	    //PathData - command - cmdParameters - bufferMode
	    IF #tempPathDataCmd_checking.cmdParameters.bufferMode <> "BM_BUFFERED"
	      AND #tempPathDataCmd_checking.cmdParameters.bufferMode <> "BM_BLENDING_LOW"
	      AND #tempPathDataCmd_checking.cmdParameters.bufferMode <> "BM_BLENDING_HIGH"
	    THEN
	      #LKinCtrl_CheckPathDataCmd := #ERR_PATHDATA_BUFFERMODE;
	      RETURN;
	    END_IF;
	    
	    //PathData - command - cmdParameters - dynamicAdaption
	    IF #tempPathDataCmd_checking.cmdParameters.dynamicAdaption > "DA_WITH_CONSTANT_LIMITS"
	    THEN
	      #LKinCtrl_CheckPathDataCmd := #ERR_PATHDATA_DYNAMICADAPTION;
	      RETURN;
	    END_IF;
	    
	    //PathData - command - setFlags
	    FOR #tempFlagCtr := 1 TO "LKINCTRL_NO_OF_CMD_SETFLAGS" DO
	      // check flag to be in range of flags InOut array at LKinCtrl_MC_MovePath
	      IF #tempPathDataCmd_checking.setFlags[#tempFlagCtr].flag <> -1
	        AND (#tempPathDataCmd_checking.setFlags[#tempFlagCtr].flag < #firstFlag OR #tempPathDataCmd_checking.setFlags[#tempFlagCtr].flag > #lastFlag)
	      THEN
	        #LKinCtrl_CheckPathDataCmd := #ERR_PATHDATA_SETFLAGS_FLAG;
	        RETURN;
	      END_IF;
	      
	      // check flagMode to be valid
	      IF "LKinCtrl_CheckFlagMode"(#tempPathDataCmd_checking.setFlags[#tempFlagCtr].flagMode) = FALSE THEN
	        #LKinCtrl_CheckPathDataCmd := #ERR_PATHDATA_SETFLAGS_FLAGMODE;
	        RETURN;
	      END_IF;
	    END_FOR;
	    
	    //PathData - command - valueFlags
	    FOR #tempFlagCtr := 1 TO "LKINCTRL_NO_OF_CMD_VALUEFLAGS" DO
	      // check flag to be in range of flags InOut array at LKinCtrl_MC_MovePath
	      IF #tempPathDataCmd_checking.valueFlags[#tempFlagCtr].flag <> -1
	        AND (#tempPathDataCmd_checking.valueFlags[#tempFlagCtr].flag < #firstFlag OR #tempPathDataCmd_checking.valueFlags[#tempFlagCtr].flag > #lastFlag)
	      THEN
	        #LKinCtrl_CheckPathDataCmd := #ERR_PATHDATA_VALUEFLAGS_FLAG;
	        RETURN;
	      END_IF;
	      
	      // check flagMode to be valid
	      IF "LKinCtrl_CheckFlagMode"(#tempPathDataCmd_checking.valueFlags[#tempFlagCtr].flagMode) = FALSE THEN
	        #LKinCtrl_CheckPathDataCmd := #ERR_PATHDATA_VALUEFLAGS_FLAGMODE;
	        RETURN;
	      END_IF;
	    END_FOR;
	  END_REGION
	END_REGION CHECK_COMMAND
	
	
END_FUNCTION

FUNCTION "LKinCtrl_CheckFlagMode" : Bool
TITLE = LKinCtrl_CheckFlagMode
{ S7_Optimized_Access := 'TRUE' }
AUTHOR : 'handling.team.automation@siemens.com'
FAMILY : LKinCtrl
VERSION : 5.0
//Check given flag mode to be valid
   VAR_INPUT 
      flagMode : DInt;   // Flagmode input
   END_VAR


BEGIN
	//==========================================================================================
	// SIEMENS AG
	// (c)Copyright 2022 All Rights Reserved
	//------------------------------------------------------------------------------------------
	// Library: LKinCtrl
	// Tested with: S7-1517T-3 PN/DP
	// Engineering: TIA Portal V18
	// Restrictions: ---
	// Requirements: S7-1500T FW 3.0
	// Functionality: LKinCtrl_CheckFlagMode
	// The FC checks FlagMode of command to be configured correctly
	//
	// Support: tech.team.motioncontrol@siemens.com
	// Note: Parameter comments are only available in language 'English (United States)'
	//------------------------------------------------------------------------------------------
	// Change log table:
	// Version    Date          Expert in charge    Changes applied
	// 01.00.00   21.12.2022    FR                  First release version v1.0
	//===========================================================================================
	
	CASE #flagMode OF
	  "LKINCTRL_FM_DEACTIVATED", // 0
	  "LKINCTRL_FM_SET_BEFORE_AND_NO_RESET", // 1
	  "LKINCTRL_FM_SET_BEFORE_AND_RESET_AFTER", // 2
	  "LKINCTRL_FM_SET_BEFORE_AND_RESET_AFTER_ONE_CYCLE", // 3
	  "LKINCTRL_FM_SET_BEFORE_AND_NO_RESET_AND_WAIT_FOR_ACKNOWLEDGE", // 5
	  "LKINCTRL_FM_SET_AT_REMAINING_DISTANCE", // 10
	  "LKINCTRL_FM_SET_AFTER_AND_NO_RESET", // 11
	  "LKINCTRL_FM_SET_AFTER_AND_RESET_AFTER_ONE_CYCLE", // 13
	  "LKINCTRL_FM_SET_AFTER_AND_NO_RESET_AND_WAIT_FOR_ACKNOWLEDGE", // 15
	  "LKINCTRL_FM_RESET_BEFORE", // 20
	  "LKINCTRL_FM_RESET_AFTER", // 21
	  "LKINCTRL_FM_RESET_AT_REMAINING_DISTANCE", // 22
	  "LKINCTRL_FM_NO_SET_AND_WAIT_FOR_FALSE_ONCE", // 25
	  "LKINCTRL_FM_NO_SET_AND_WAIT_FOR_TRUE_ONCE": // 26
	    #LKinCtrl_CheckFlagMode := TRUE; // FlagMode ok
	  ELSE  // not a valid mode
	    #LKinCtrl_CheckFlagMode := FALSE;
	END_CASE;
	
	
END_FUNCTION

FUNCTION "LKinCtrl_CheckUserFrame" : Bool
TITLE = LKinCtrl_CheckUserFrame
{ S7_Optimized_Access := 'TRUE' }
AUTHOR : 'handling.team.automation@siemens.com'
FAMILY : LKinCtrl
VERSION : 5.0
//Checks a command if it can be executed with a user frame
   VAR_INPUT 
      cmdType : DInt;
      coordinateSystem : DInt;
      circMode : DInt;
      userFrames : Array["LKINCTRL_CS_NO_OF_FIRST_USER_FRAME".."LKINCTRL_CS_NO_OF_LAST_USER_FRAME"] of "LKinCtrl_typeFrame";
   END_VAR

   VAR_TEMP 
      tempReturnValue : Bool;
   END_VAR


BEGIN
	//==========================================================================================
	// SIEMENS AG
	// (c)Copyright 2021 All Rights Reserved
	//------------------------------------------------------------------------------------------
	// Library: LKinCtrl
	// Tested with: S7-1517T-3 PN/DP
	// Engineering: TIA Portal V16
	// Restrictions: ---
	// Requirements: S7-1500T FW 2.8
	// Functionality: LKinCtrl_CheckUserFrame
	// The FC checks a given command if it can be executed with a user frame
	//
	// Support: tech.team.motioncontrol@siemens.com
	// Note: Parameter comments are only available in language 'English (United States)'
	//------------------------------------------------------------------------------------------
	// Change log table:
	// Version    Date          Expert in charge    Changes applied
	// 01.00.00   20.08.2021    FR                  First released version
	//===========================================================================================
	
	// Initialize temporary return value
	#tempReturnValue := FALSE;
	
	IF #coordinateSystem >= "LKINCTRL_CS_NO_OF_FIRST_USER_FRAME"
	    AND #coordinateSystem <= "LKINCTRL_CS_NO_OF_LAST_USER_FRAME"
	THEN
	    // Check if circular command is used
	    IF (#cmdType = "LKINCTRL_MC_MOVECIRCULARABS" OR #cmdType = "LKINCTRL_MC_MOVECIRCULARREL")
	        AND (#circMode <> "CM_BORDER")
	    THEN
	        // Check if used frame has a rotation
	        IF #userFrames[#coordinateSystem].a <> 0.0
	            OR #userFrames[#coordinateSystem].b <> 0.0
	            OR #userFrames[#coordinateSystem].c <> 0.0
	        THEN
	            // Command is not allowed! --> Not OK
	            #tempReturnValue := FALSE;
	        ELSE
	            // No rotation in user frame --> OK
	            #tempReturnValue := TRUE;
	        END_IF;
	    ELSE
	        // Not a critical circular command --> OK
	        #tempReturnValue := TRUE;
	    END_IF;
	ELSE
	    // Command is not executed in user CS -> OK
	    #tempReturnValue := TRUE;
	END_IF;
	
	
	// Write return value
	#LKinCtrl_CheckUserFrame := #tempReturnValue;
	
	
	
	
	
	
END_FUNCTION

FUNCTION "LKinCtrl_ConvElements_PathDataToPathData_PreBuf" : Void
TITLE = LKinCtrl_ConvElements_PathDataToPathData_PreBuf
{ S7_Optimized_Access := 'TRUE' }
AUTHOR : 'handling.team.automation@siemens.com'
FAMILY : LKinCtrl
VERSION : 5.0
//The FC converts PathData commands to elements fitting the PathData_PreBuf structure
   VAR_INPUT 
      copyCompensatedParametes : Bool;   // copy selection compensated parameters
      copyTransitionParameters : Bool;   // copy selection transition parameters
      copyFlags : Bool;   // copy selection flags
   END_VAR

   VAR_IN_OUT 
      pathDataElement : "LKinCtrl_typePathDataElement";   // in: pathDataElement to be copied
      pathDataPreBufElement : "LKinCtrl_typePathDataElement_PreBuf";   // out: pathDataElement_PreBuf to be written
      pathDataName : String;   // name of PathData to be copied (separate from element)
   END_VAR

   VAR_TEMP 
      tempFlagCtr : Int;
   END_VAR


BEGIN
	//==========================================================================================
	// SIEMENS AG
	// (c)Copyright 2019 All Rights Reserved
	//------------------------------------------------------------------------------------------
	// Library: LKinCtrl
	// Tested with: S7-1517T-3 PN/DP
	// Engineering: TIA Portal V15
	// Restrictions: ---
	// Requirements: S7-1500T FW 2.5
	// Functionality: LKinCtrl_ConvElements_PathDataToPathData_PreBuf
	// The FC converts PathData commands to elements fitting the PathData_PreBuf structure
	//
	// Support: tech.team.motioncontrol@siemens.com
	// Note: Parameter comments are only available in language 'English (United States)'
	//------------------------------------------------------------------------------------------
	// Change log table:
	// Version    Date          Expert in charge    Changes applied
	// 01.00.00   20.02.2019    JR                  First release version v1.0
	// 01.00.01   16.08.2019    JR                  added setFlags edit code: flagMode: 3 -> 2
	// 01.00.02   28.01.2020    FR                  added value flags to copyFlags
	// 01.01.00   04.03.2021    FR                  added all cmd parameters
	// 01.01.01   03.01.2024    SF                  added PickAndPlace parameters
	//===========================================================================================
	
	// General info
	#pathDataPreBufElement.pathDataName := #pathDataName;
	#pathDataPreBufElement.cmdType := #pathDataElement.cmdType;
	#pathDataPreBufElement.cmdName := #pathDataElement.cmdName;
	
	
	// Target coordinates / circle parameter
	IF #copyCompensatedParametes THEN // copy target positions
	    #pathDataPreBufElement.cmdCoordinates.targetPosition[1] := #pathDataElement.cmdCoordinates.cartesianPosition.x;
	    #pathDataPreBufElement.cmdCoordinates.targetPosition[2] := #pathDataElement.cmdCoordinates.cartesianPosition.y;
	    #pathDataPreBufElement.cmdCoordinates.targetPosition[3] := #pathDataElement.cmdCoordinates.cartesianPosition.z;
	    #pathDataPreBufElement.cmdCoordinates.targetPosition[4] := #pathDataElement.cmdCoordinates.cartesianPosition.a;
	    #pathDataPreBufElement.cmdCoordinates.targetPosition[5] := #pathDataElement.cmdCoordinates.cartesianPosition.b;
	    #pathDataPreBufElement.cmdCoordinates.targetPosition[6] := #pathDataElement.cmdCoordinates.cartesianPosition.c;
	    #pathDataPreBufElement.cmdCoordinates.coordSystem := #pathDataElement.cmdCoordinates.coordSystem;
	    
	    #pathDataPreBufElement.cmdParameters.circleParameters := #pathDataElement.cmdParameters.circleParameters;
	END_IF;
	
	// Cmd parameter - general
	#pathDataPreBufElement.cmdParameters.pathDynamics := #pathDataElement.cmdParameters.pathDynamics;
	#pathDataPreBufElement.cmdParameters.orientationDynamics := #pathDataElement.cmdParameters.orientationDynamics;
	#pathDataPreBufElement.cmdParameters.orientationDirection := #pathDataElement.cmdParameters.orientationDirection;
	#pathDataPreBufElement.cmdParameters.dynamicAdaption := #pathDataElement.cmdParameters.dynamicAdaption;
	#pathDataPreBufElement.cmdParameters.toolNumber := #pathDataElement.cmdParameters.toolNumber;
	#pathDataPreBufElement.cmdParameters.bufferMode := #pathDataElement.cmdParameters.bufferMode;
	#pathDataPreBufElement.cmdParameters.conveyorParameters := #pathDataElement.cmdParameters.conveyorParameters;
	#pathDataPreBufElement.cmdParameters.moveDirectParameters := #pathDataElement.cmdParameters.moveDirectParameters;
	#pathDataPreBufElement.cmdParameters.offsetParameters := #pathDataElement.cmdParameters.offsetParameters;
	#pathDataPreBufElement.cmdParameters.zoneParameters := #pathDataElement.cmdParameters.zoneParameters;
	#pathDataPreBufElement.cmdParameters.pickAndPlaceParameters := #pathDataElement.cmdParameters.pickAndPlaceParameters;
	
	//Measurement Cmd
	#pathDataPreBufElement.measurementCmd := #pathDataElement.measurementCmd;
	
	// Transition parameter
	IF #copyTransitionParameters THEN
	    #pathDataPreBufElement.cmdParameters.transitionParameters := #pathDataElement.cmdParameters.transitionParameters;
	END_IF;
	
	// Flags
	IF #copyFlags THEN
	    // ---------------------------------------------------------------
	    // Set flags (bool)
	    // ---------------------------------------------------------------
	    #pathDataPreBufElement.setFlags := #pathDataElement.setFlags;
	    // change flagMode 3 to flagMode 2 as functionality is equal
	    // check for cmd to be flagOnly cmd
	    // check for cmd to implement flag and flagMode to be flagMode 3
	    FOR #tempFlagCtr := 1 TO "LKINCTRL_NO_OF_CMD_SETFLAGS" DO
	        IF #pathDataPreBufElement.cmdType = "LKINCTRL_CMD_FLAG_ONLY"
	            AND #pathDataPreBufElement.setFlags[#tempFlagCtr].flag <> -1
	            AND #pathDataPreBufElement.setFlags[#tempFlagCtr].flagMode = "LKINCTRL_FM_SET_BEFORE_AND_RESET_AFTER_ONE_CYCLE"
	        THEN
	            // change flagMode to flagMode 2
	            #pathDataPreBufElement.setFlags[#tempFlagCtr].flagMode := "LKINCTRL_FM_SET_BEFORE_AND_RESET_AFTER";
	        END_IF;
	    END_FOR;
	    // ---------------------------------------------------------------
	    
	    // ---------------------------------------------------------------
	    // Value flags (LReal)
	    // ---------------------------------------------------------------
	    #pathDataPreBufElement.valueFlags := #pathDataElement.valueFlags;
	    // change flagMode 3 to flagMode 2 as functionality is equal
	    // check for cmd to be flagOnly cmd
	    // check for cmd to implement flag and flagMode to be flagMode 3
	    FOR #tempFlagCtr := 1 TO "LKINCTRL_NO_OF_CMD_VALUEFLAGS" DO
	        IF #pathDataPreBufElement.cmdType = "LKINCTRL_CMD_FLAG_ONLY"
	            AND #pathDataPreBufElement.valueFlags[#tempFlagCtr].flag <> -1
	            AND #pathDataPreBufElement.valueFlags[#tempFlagCtr].flagMode = "LKINCTRL_FM_SET_BEFORE_AND_RESET_AFTER_ONE_CYCLE"
	        THEN
	            // change flagMode to flagMode 2
	            #pathDataPreBufElement.valueFlags[#tempFlagCtr].flagMode := "LKINCTRL_FM_SET_BEFORE_AND_RESET_AFTER";
	        END_IF;
	    END_FOR;
	    // ---------------------------------------------------------------
	END_IF;
	
END_FUNCTION

FUNCTION "LKinCtrl_OffsetContour" : "LKinCtrl_typeCOffReturn"
TITLE = LKinCtrl_OffsetContour
{ S7_Optimized_Access := 'TRUE' }
AUTHOR : 'handling.team.automation@siemens.com'
FAMILY : LKinCtrl
VERSION : 5.0
//The function calculates a contour offset of a path (tool length and radius) 
   VAR_INPUT 
      toolLength : LReal;   // Tool length
      toolRadius : LReal;   // Tool radius
      pathPlane : Int;   // Path plane: XZ= 0, YZ=1, XY= 2
      compensationDirection : Int;   // Tool radius compensation direction: left=1, right = 0
   END_VAR

   VAR_IN_OUT 
      currentPosIn : "LKinCtrl_typeCOffInCurrentPos";   // Source data - current position
      nextCommandIn : "LKinCtrl_typePathDataElement";   // Source data - next command
      nextButOneCommandIn : "LKinCtrl_typePathDataElement";   // Source data - next but one command
      nextCommandOut : "LKinCtrl_typePathDataElement";   // Target data - next command
      intermediateCommandOut : "LKinCtrl_typePathDataElement";   // Target data - intermediate (additional) command
      nextButOneCommandOut : "LKinCtrl_typeCOffOutNextButOneCmd";   // Target data - next but one command
      nextPositionAbsoluteOut : "LKinCtrl_typeCartesianPosition";   // Source data - next absolute position
      nextPositionAbsoluteRadCompOut : "LKinCtrl_typeCartesianPosition";   // Source data - next absolute position (radius compensated)
   END_VAR

   VAR_TEMP 
      internalNumber : DInt;   // Internal error position
      boCmdInPathPlane : Bool;   // Command in path plane
      pathDataDelete : "LKinCtrl_typeCOffPathDataOut" := (((), (), (), (), (), (((), (), (), (), (), ()), ()), (((), (), (), ()), ((), (), (), ()), (), (), [-1.0], (), (), ((), (), [()]), ((), ()), (()), ((), (), [()], (), (), (), ()), ((), (), ()), (([()], (), (), ()), ([()], (), (), ()))), [((), (), ()), ((), (), ()), ((), (), ())], [((), (), (), ()), ((), (), (), ()), ((), (), (), ()), ((), (), (), ())], [6(TRUE)]), ((), (), (), (), (), (((), (), (), (), (), ()), ()), (((), (), (), ()), ((), (), (), ()), (), (), [-1.0], (), (), ((), (), [()]), ((), ()), (()), ((), (), [()], (), (), (), ()), ((), (), ()), (([()], (), (), ()), ([()], (), (), ()))), [((), (), ()), ((), (), ()), ((), (), ())], [((), (), (), ()), ((), (), (), ()), ((), (), (), ()), ((), (), (), ())], [6(TRUE)]), ([()]), ((), (), (), (), (), ()), ((), (), (), (), (), ()));   // Delete data structure
      tempCurrentPoint : "LKinCtrl_typeCOff3DPoint";   // End point 1st command - current command
      tempCurrentPointPathPlane : "LKinCtrl_typeCOff3DPoint";   // End point 1st command - current command - path plane
      tempCurrentPointRadComp : "LKinCtrl_typeCOff3DPoint";   // End point 1st command - current command - radius compensated
      tempNextCmdIn : "LKinCtrl_typeCOffCmdInInternal";   // Next command input
      tempNextButOneCmdIn : "LKinCtrl_typeCOffCmdInInternal";   // Next but one command input
      tempNextCmdOut : "LKinCtrl_typeCOffCmdOutInternal";   // Next command output
      tempIntermediateCmdOut : "LKinCtrl_typeCOffCmdOutInternal";   // Intermediate command output
      tempNextButOneCmdOut : "LKinCtrl_typeCOffCmdOutInternal";   // Next but one command output
      tempToolRadiusComp : Bool;   // TRUE: tool radius compensation used
      tempToolLengthComp : Bool;   // TRUE: tool length compensation used
      tempRetValue : Word;   // Return value
      tempMuA : LReal;
      tempMuB : LReal;
      tempCornerType : Int;
      tempPa : "LKinCtrl_typeCOff3DPoint";
      tempPb : "LKinCtrl_typeCOff3DPoint";
      tempDistance1 : LReal;
      tempDistance2 : LReal;
      tempCircleDistance1 : LReal;
      tempCircleDistance2 : LReal;
      tempCircleDistance3 : LReal;
      tempAngle : LReal;
      tempMod : DInt;
      tempPathChoice : DInt;
      tempNextCmdEndPointLevelled : "LKinCtrl_typeCOff3DPoint";
      tempNextCmdIntermediatePointLevelled : "LKinCtrl_typeCOff3DPoint";
      tempNextButOneStartPointOrthShiftedLevelled : "LKinCtrl_typeCOff3DPoint";
      tempNextButOneCmdStartPointOrthTangShiftedLevelled : "LKinCtrl_typeCOff3DPoint";
      tempNextCmdStartPointOrhtShiftLevelled : "LKinCtrl_typeCOff3DPoint";
      tempDirectionUncompensatedVec : "LKinCtrl_typeCOff3DPoint";
      tempDirectionCompensatedVec : "LKinCtrl_typeCOff3DPoint";
      tempDirectionUncompensatedUnitVec : "LKinCtrl_typeCOff3DPoint";
      tempDirectionCompensatedUnitVec : "LKinCtrl_typeCOff3DPoint";
      tempLengthCompensatedPointDifferenceVec : LReal;
   END_VAR

   VAR CONSTANT 
      COFF_TRANSITION_TOLERANCE : LReal := 0.2;   // Tolerance for additional circle - outer corner
      ERR_COFF_INVALID_TOOL_LENGTH : Word := 16#8301;   // Error - invalid tool length
      ERR_COFF_INVALID_TOOL_RADIUS : Word := 16#8302;   // Error - invalid tool radius
      ERR_COFF_INVALID_PATH_PLANE : Word := 16#8303;   // Error - invalid path plane
      ERR_COFF_INVALID_COMPENSATION_DIRECTION : Word := 16#8304;   // Error - invalid compensation direction
      ERR_COFF_FUNCTION_NOT_SUPPORTED : Word := 16#8305;   // Error - functionality not supported
      ERR_COFF_INVALID_COMMAND_TYPE : Word := 16#8306;   // Error - invalid command type
      ERR_COFF_INVALID_CIRCLE_MODE : Word := 16#8307;   // Error - invalid circle mode
      ERR_COFF_INVALID_PATH_PLANE_OF_CIRCULAR_CMD : Word := 16#8308;   // Error - invalid path plane of a circular command
      ERR_COFF_INVALID_PATH_CHOICE_OF_CIRCULAR_CMD : Word := 16#8309;   // Error - invalid path choice of circular command
      ERR_COFF_INTERNAL : Word := 16#830F;   // Error - internal
      ERR_COFF_VECTOR_LENGTH_ZERO : Word := 16#8310;   // Error - vector length is zero
      ERR_COFF_INVALID_ACOS_ARGUMENT : Word := 16#8311;   // Error - invalid ACOS argument
      ERR_COFF_LINES_DO_NOT_INTERSECT : Word := 16#8312;   // Error - no solution, lines don't intersect
      ERR_COFF_ZERO_VECTOR : Word := 16#8313;   // Error - zero vector
      ERR_COFF_CMD_LENGTH_ZERO : Word := 16#8314;   // Error - cmd with length zero not permitted
      ERR_COFF_LINE_CIRCLE_DO_NOT_INTERSECT : Word := 16#8315;   // Error - no solution - line and circle don't intersect
      ERR_COFF_CIRCLES_DO_NOT_INTERSECT : Word := 16#8318;   // Error - no solution - circles don't intersect
      ERR_COFF_ONE_CIRC_CONTAINED_IN_THE_OTHER : Word := 16#8319;   // Error - one circle is contained in the other
      ERR_COFF_NO_SOLUTION_FOR_GIVEN_LINEAR_CMD : Word := 16#8320;   // Error - no valid solution with given linear command
      ERR_COFF_NO_SOLUTION_FOR_GIVEN_CIRCULAR_CMD : Word := 16#8321;   // Error - no valid solution with given circular command
      ERR_COFF_LINEAR_CMD_AND_TOOL_RADIUS_LEAD_TO_REVERSAL : Word := 16#8322;   // Error - linear command in combination with tool radius leads to reversal movement
      ERR_COFF_CIRCLE_CENTERS_EQUAL : Word := 16#8350;   // Error - circle centers are equal infinite intersections (only internal)
      COFF_REGION_TYPE_NONE : Int := 0;   // Region type: none
      COFF_REGION_TYPE_PLAUSIBILITY : Int := 1;   // Region type: plausibitlity general
      COFF_REGION_TYPE_PLAUSIBILITY_NEXT_CMD : Int := 2;   // Region type: plausibility next command
      COFF_REGION_TYPE_PLAUSIBILITY_NEXT_BUT_ONE_CMD : Int := 3;   // Region type: plausibility next but one command
      COFF_REGION_TYPE_PRE_CALC : Int := 4;   // Region type: precalculation
      COFF_REGION_TYPE_RAD_COMP_NEXT_CMD_LIN : Int := 5;   // Region type: radius compensation next command linear
      COFF_REGION_TYPE_RAD_COMP_LIN_LIN : Int := 6;   // Region type: radius compensation next command linear, next but one command linear
      COFF_REGION_TYPE_RAD_COMP_LIN_CIRC : Int := 7;   // Region type: radius compensation next command linear, next but one command circular
      COFF_REGION_TYPE_RAD_COMP_LIN_NONE : Int := 8;   // Region type: radius compensation next command linear, next but one command none
      COFF_REGION_TYPE_RAD_COMP_LIN_GEN : Int := 9;   // Region type: radius compensation next command linear - general
      COFF_REGION_TYPE_RAD_COMP_NEXT_CMD_CIRC : Int := 10;   // Region type: radius compensation next command circular
      COFF_REGION_TYPE_RAD_COMP_CIRC_LIN : Int := 11;   // Region type: radius compensation next command circular next but one command linear
      COFF_REGION_TYPE_RAD_COMP_CIRC_CIRC : Int := 12;   // Region type: radius compensation next command circular, next but one command circular
      COFF_REGION_TYPE_RAD_COMP_CIRC_NONE : Int := 13;   // Region type: radius compensation next command circular, next but one command none
      COFF_REGION_TYPE_RAD_COMP_CIRC_GEN : Int := 14;   // Region type: radius compensation next command circular - general
      COFF_REGION_TYPE_LEN_COMP_NEXT : Int := 15;   // Region type: tool length compensation next command
      COFF_REGION_TYPE_LEN_COMP_INTER_CMD : Int := 16;   // Region type: tool length compensation intermediate command
      COFF_REGION_TYPE_LEN_COMP_NEXT_BUT_ONE_CMD : Int := 17;   // Region type: tool length compensation next but one command
      COFF_REGION_TYPE_OUTPUT_DATA : Int := 18;   // Region type: ouptut data
      COFF_TOLERANCE : LReal := 0.001;   // Tolerance
      RADIUS_PLAUSIBLITY_TOLERANCE : LReal := 0.1;   // Radius tolerance
      COFF_CIRC_REVERSAL_TOLERANCE_ANGLE : LReal := 90.0;   // Reversal tolerance check for circle
   END_VAR


BEGIN
	//==========================================================================================
	// SIEMENS AG
	// (c)Copyright 2019 All Rights Reserved
	//------------------------------------------------------------------------------------------
	// Library: LKinCtrl
	// Tested with: S7-1515T-3 PN/DP
	// Engineering: TIA Portal V15
	// Restrictions: ---
	// Requirements: S7-1500T FW 2.5
	// Functionality: LKinCtrl_OffsetContour
	// The function calculates a contour offset of a path (tool length and radius) 
	// Support: tech.team.motioncontrol@siemens.com
	// Note: Parameter comments are only available in language 'English (United States)'
	//------------------------------------------------------------------------------------------
	// Change log table:
	// Version    Date          Expert in charge    Changes applied
	// 00.09.00   2019-02-06    AW                  Beta version
	// 01.00.00   2019-03-08    AW                  First release version
	// 01.01.00   2020-08-14    AW                  Bug fix - intersection point of 1st and 2nd circle (equal circle centers)
	//                                                       - LKinCtrl_CalcLineCircleIntersectionPoint
	//                                                       - LKinCtrl_CalcCircleCircleIntersectionPoint
	//                                              length compensation (circle with radius and endpoint)
	// 01.01.01  2020-08-25     AW                  Additional tolerance intersection of two circles (possible tiny floating point
	//                                              deviations in case of one intersection point) - LKinCtrl_CalcCircleCircleIntersectionPoint
	// 01.01.02  2020-10-13     AW                  fix - check innter outer corner - not done for linear commands in same direction anymore
	//                                              additional check for next command LINEAR and next but one command NONE
	//                                              avoid reversal movement for small linear path length in combination with big compensation radius
	// 01.01.03  2020-11-09     AW                  bugfix addtional check - N E X T   B U T   O N E   C M D  -  N O N E                                          
	// 01.02.00  2021-03-11     FR                  changed interface to reduce nesting depth
	// 01.02.01  2021-11-12     AW                  bugfix intersection point of 1st linear and 2nd circular command
	// 01.02.02  2022-05-19     AW                  bugfix M O D I F Y   N E X T   C I R C U L A R   C O M M A N D - CIRC_CENTER - calculate compensated angle,
	//                                              additional plausibility check - 
	//                                              tool radius must not be greater than circle radius
	//                                              tool radius must not be greater than circle start and end point (uncompensated)
	//                                              new constant: RADIUS_PLAUSIBLITY_TOLERANCE
	//===========================================================================================
	
	// Plausibility checks of parameter
	REGION PLAUSIBILITY_CHECK
	  // Check tool length
	  IF (#toolLength < 0.0)
	  THEN
	    #LKinCtrl_OffsetContour.returnValue := #ERR_COFF_INVALID_TOOL_LENGTH; // Invalid tool length
	    #LKinCtrl_OffsetContour."region" := #COFF_REGION_TYPE_PLAUSIBILITY;
	    #LKinCtrl_OffsetContour.internalNumber := 101;
	    RETURN;
	    
	    // Check tool radius  
	  ELSIF (#toolRadius < 0.0)
	  THEN
	    #LKinCtrl_OffsetContour.returnValue := #ERR_COFF_INVALID_TOOL_RADIUS; // Invalid tool radius
	    #LKinCtrl_OffsetContour."region" := #COFF_REGION_TYPE_PLAUSIBILITY;
	    #LKinCtrl_OffsetContour.internalNumber := 102;
	    RETURN;
	  END_IF;
	  
	  // Check circular path plane in combination with global path plane - next command
	  IF ((((#nextCommandIn.cmdType = "LKINCTRL_MC_MOVECIRCULARABS") OR
	    (#nextCommandIn.cmdType = "LKINCTRL_MC_MOVECIRCULARREL")) AND
	    ((#nextCommandIn.cmdParameters.circleParameters.circMode = "CM_CENTER") OR
	    (#nextCommandIn.cmdParameters.circleParameters.circMode = "CM_RADIUS")) AND
	    (#pathPlane <> #nextCommandIn.cmdParameters.circleParameters.circlePlane)))
	  THEN
	    #LKinCtrl_OffsetContour.returnValue := #ERR_COFF_INVALID_PATH_PLANE_OF_CIRCULAR_CMD; // Invalid path plane of a circular command
	    #LKinCtrl_OffsetContour."region" := #COFF_REGION_TYPE_PLAUSIBILITY_NEXT_CMD;
	    #LKinCtrl_OffsetContour.internalNumber := 103;
	    RETURN;
	  END_IF;
	  
	  // Check circular path plane in combination with global path plane - next but one command
	  IF ((((#nextButOneCommandIn.cmdType = "LKINCTRL_MC_MOVECIRCULARABS") OR
	    (#nextButOneCommandIn.cmdType = "LKINCTRL_MC_MOVECIRCULARREL")) AND
	    ((#nextButOneCommandIn.cmdParameters.circleParameters.circMode = "CM_CENTER") OR
	    (#nextButOneCommandIn.cmdParameters.circleParameters.circMode = "CM_RADIUS")) AND
	    (#pathPlane <> #nextButOneCommandIn.cmdParameters.circleParameters.circlePlane)))
	  THEN
	    #LKinCtrl_OffsetContour.returnValue := #ERR_COFF_INVALID_PATH_PLANE_OF_CIRCULAR_CMD; // Invalid path plane of a circular command
	    #LKinCtrl_OffsetContour."region" := #COFF_REGION_TYPE_PLAUSIBILITY_NEXT_BUT_ONE_CMD;
	    #LKinCtrl_OffsetContour.internalNumber := 104;
	    RETURN;
	  END_IF;
	  
	  // Tool radius compensation?
	  #tempToolRadiusComp := FALSE;
	  IF (#toolRadius > 0.0)
	  THEN
	    // Check path plane
	    IF ((#pathPlane >= "CP_XZ") AND (#pathPlane <= "CP_XY"))
	    THEN
	      IF ((#compensationDirection >= "LKINCTRL_COMP_LEFT") AND (#compensationDirection <= "LKINCTRL_COMP_RIGHT"))
	      THEN
	        #tempToolRadiusComp := TRUE;
	      ELSE
	        #LKinCtrl_OffsetContour.returnValue := #ERR_COFF_INVALID_COMPENSATION_DIRECTION; // Invalid compensation direction
	        #LKinCtrl_OffsetContour."region" := #COFF_REGION_TYPE_PLAUSIBILITY;
	        #LKinCtrl_OffsetContour.internalNumber := 105;
	        RETURN;
	      END_IF;
	    ELSE
	      #LKinCtrl_OffsetContour.returnValue := #ERR_COFF_INVALID_PATH_PLANE; // Invalid path plane
	      #LKinCtrl_OffsetContour."region" := #COFF_REGION_TYPE_PLAUSIBILITY;
	      #LKinCtrl_OffsetContour.internalNumber := 106;
	      RETURN;
	    END_IF;
	  END_IF;
	  
	  // Tool length compensation=
	  IF (#toolLength > 0.0)
	  THEN
	    #tempToolLengthComp := TRUE;
	  ELSE
	    #tempToolLengthComp := FALSE;
	  END_IF;
	END_REGION PLAUSIBILITY_CHECK
	
	
	REGION Delete data
	  //#pathDataOut := #pathDataDelete;
	  #nextCommandOut := #pathDataDelete.nextCommand;
	  #intermediateCommandOut := #pathDataDelete.intermediateCommand;
	  #nextButOneCommandOut := #pathDataDelete.nextButOneCommand;
	  #nextPositionAbsoluteOut := #pathDataDelete.nextPositionAbsolute;
	  #nextPositionAbsoluteRadCompOut := #pathDataDelete.nextPositionAbsoluteRadComp;
	END_REGION
	
	REGION General
	  
	  IF (#tempToolRadiusComp OR #tempToolLengthComp) THEN
	    // Output data preliminary
	    // Next command
	    #nextCommandOut := #nextCommandIn;
	    // Current position
	    // --------------------------
	    #tempCurrentPoint := "LKinCtrl_CartesianCoordTo3DPoint"(#currentPosIn.positionAbsolute);
	    #tempCurrentPointRadComp := "LKinCtrl_CartesianCoordTo3DPoint"(#currentPosIn.positionAbsoluteRadComp);
	    
	    // Next command
	    // --------------------------
	    #tempNextCmdIn.cmdType := #nextCommandIn.cmdType;
	    // Write to output data - modifications done later
	    #tempNextCmdOut.cmdType := #tempNextCmdIn.cmdType;
	    
	    #tempNextCmdIn.transitionParameter1 := #nextCommandIn.cmdParameters.transitionParameters[1];
	    #tempNextCmdIn.bufferMode := #nextCommandIn.cmdParameters.bufferMode;
	    
	    IF ((#tempNextCmdIn.cmdType = "LKINCTRL_MC_MOVELINEARABS") OR
	      (#tempNextCmdIn.cmdType = "LKINCTRL_MC_MOVELINEARREL"))
	    THEN
	      IF (#tempNextCmdIn.cmdType = "LKINCTRL_MC_MOVELINEARABS") THEN
	        // Absolute coordinates
	        // End point is defined
	        
	        #tempNextCmdIn.endPoint := "LKinCtrl_CartesianCoordTo3DPoint"(cartesianCoord := #nextCommandIn.cmdCoordinates.cartesianPosition);
	        
	      ELSIF (#tempNextCmdIn.cmdType = "LKINCTRL_MC_MOVELINEARREL") THEN
	        // Relative coordinates -> calculate absolute coordinate
	        #tempNextCmdIn.endPoint := "LKinCtrl_VecAdd"(vIn1 := #tempCurrentPoint,
	                                                     vIn2 := "LKinCtrl_CartesianCoordTo3DPoint"(#nextCommandIn.cmdCoordinates.cartesianPosition));
	        
	        // Set command type to absolute
	        #tempNextCmdOut.cmdType := "LKINCTRL_MC_MOVELINEARABS";
	      END_IF;
	      
	      // Check if cmd length is unequal zero
	      IF ("LKinCtrl_VecAbs"("LKinCtrl_VecSub"(vIn1 := #tempCurrentPoint, vIn2 := #tempNextCmdIn.endPoint)) < #COFF_TOLERANCE) THEN
	        
	        // Not allowed - function has no memory and therefore can't treat a command length of zero correctly
	        #LKinCtrl_OffsetContour.returnValue := #ERR_COFF_CMD_LENGTH_ZERO;
	        #LKinCtrl_OffsetContour."region" := #COFF_REGION_TYPE_PLAUSIBILITY_NEXT_CMD;
	        #LKinCtrl_OffsetContour.internalNumber := 201;
	        RETURN;
	      END_IF;
	      
	      // Check if next linear command has at least one component in path plane direction
	      #tempRetValue := "LKinCtrl_CalcVecDistancePathPlane"(vectorInA := #tempCurrentPoint,
	                                                           vectorInB := #tempNextCmdIn.endPoint,
	                                                           pathPlane := #pathPlane,
	                                                           distancePathPlane => #tempDistance1);
	      
	      IF (#tempRetValue <> 0) THEN
	        #LKinCtrl_OffsetContour.returnValue := #tempRetValue;
	        #LKinCtrl_OffsetContour."region" := #COFF_REGION_TYPE_PLAUSIBILITY_NEXT_CMD;
	        #LKinCtrl_OffsetContour.subBlockNumber := 35055;
	        #LKinCtrl_OffsetContour.internalNumber := 202;
	        RETURN;
	      END_IF;
	      
	      // Check if movement is in respective path plane
	      IF (#tempDistance1 > 0.0) THEN
	        // Change current position?
	        // --------------------------
	        #boCmdInPathPlane := true;
	      ELSE
	        #boCmdInPathPlane := false;
	      END_IF;
	      
	    ELSIF ((#tempNextCmdIn.cmdType = "LKINCTRL_MC_MOVECIRCULARABS") OR
	      (#tempNextCmdIn.cmdType = "LKINCTRL_MC_MOVECIRCULARREL"))
	    THEN
	      
	      #tempNextCmdIn.circleMode := #nextCommandIn.cmdParameters.circleParameters.circMode;
	      #tempNextCmdIn.pathChoice := #nextCommandIn.cmdParameters.circleParameters.pathChoice;
	      
	      // Check for invalid path choice
	      IF ((#tempNextCmdIn.pathChoice < "PC_POSITIVE") OR
	        (#tempNextCmdIn.pathChoice > "PC_NEGATIVE"))
	      THEN
	        #LKinCtrl_OffsetContour.returnValue := #ERR_COFF_INVALID_PATH_CHOICE_OF_CIRCULAR_CMD; // Invalid path plane of a circular command
	        #LKinCtrl_OffsetContour."region" := #COFF_REGION_TYPE_PLAUSIBILITY_NEXT_CMD;
	        #LKinCtrl_OffsetContour.internalNumber := 203;
	        RETURN;
	      END_IF;
	      
	      #tempNextCmdIn.circlePlane := #nextCommandIn.cmdParameters.circleParameters.circlePlane;
	      
	      IF ((#tempNextCmdIn.circleMode = "CM_BORDER") OR
	        (#tempNextCmdIn.circleMode = "CM_RADIUS"))
	      THEN
	        // End point is defined
	        IF (#tempNextCmdIn.cmdType = "LKINCTRL_MC_MOVECIRCULARABS") THEN
	          // Absolute coordinates
	          #tempNextCmdIn.endPoint := "LKinCtrl_CartesianCoordTo3DPoint"(cartesianCoord := #nextCommandIn.cmdCoordinates.cartesianPosition);
	        ELSE
	          // Relative coordinates -> calculate absolute coordinate
	          #tempNextCmdIn.endPoint := "LKinCtrl_VecAdd"(vIn1 := #tempCurrentPoint,
	                                                       vIn2 := "LKinCtrl_CartesianCoordTo3DPoint"(#nextCommandIn.cmdCoordinates.cartesianPosition));
	        END_IF;
	        
	        IF (#tempNextCmdIn.circleMode = "CM_BORDER") THEN
	          IF (#tempNextCmdIn.cmdType = "LKINCTRL_MC_MOVECIRCULARABS") THEN
	            // Absolute coordinates
	            #tempNextCmdIn.circleIntermediatePoint.x := #nextCommandIn.cmdParameters.circleParameters.auxPoint[1];
	            #tempNextCmdIn.circleIntermediatePoint.y := #nextCommandIn.cmdParameters.circleParameters.auxPoint[2];
	            #tempNextCmdIn.circleIntermediatePoint.z := #nextCommandIn.cmdParameters.circleParameters.auxPoint[3];
	          ELSE
	            // Relative coordinates -> calculate absolute coordinate
	            #tempNextCmdIn.circleIntermediatePoint.x := #tempCurrentPoint.x + #nextCommandIn.cmdParameters.circleParameters.auxPoint[1];
	            #tempNextCmdIn.circleIntermediatePoint.y := #tempCurrentPoint.y + #nextCommandIn.cmdParameters.circleParameters.auxPoint[2];
	            #tempNextCmdIn.circleIntermediatePoint.z := #tempCurrentPoint.z + #nextCommandIn.cmdParameters.circleParameters.auxPoint[3];
	          END_IF;
	        END_IF;
	        
	        IF (#tempNextCmdIn.circleMode = "CM_RADIUS") THEN
	          #tempNextCmdIn.circleRadius := #nextCommandIn.cmdParameters.circleParameters.radius;
	          
	          // "Third" coordinate is ignored by system - also ignore here!
	          // Use start coordinate of circle instead
	          IF (#pathPlane = "CP_XZ") THEN
	            #tempNextCmdIn.endPoint.y := #tempCurrentPoint.y;
	          ELSIF (#pathPlane = "CP_YZ") THEN
	            #tempNextCmdIn.endPoint.x := #tempCurrentPoint.x;
	          ELSIF (#pathPlane = "CP_XY") THEN
	            #tempNextCmdIn.endPoint.z := #tempCurrentPoint.z;
	          END_IF;
	        END_IF;
	        
	      ELSIF (#tempNextCmdIn.circleMode = "CM_CENTER") THEN
	        #tempNextCmdIn.circleAngle := #nextCommandIn.cmdParameters.circleParameters.arc;
	        
	        IF (#tempNextCmdIn.cmdType = "LKINCTRL_MC_MOVECIRCULARABS") THEN
	          // Absolute coordinates
	          #tempNextCmdIn.circleCenterPoint.x := #nextCommandIn.cmdParameters.circleParameters.auxPoint[1];
	          #tempNextCmdIn.circleCenterPoint.y := #nextCommandIn.cmdParameters.circleParameters.auxPoint[2];
	          #tempNextCmdIn.circleCenterPoint.z := #nextCommandIn.cmdParameters.circleParameters.auxPoint[3];
	        ELSE
	          // Relative coordinates -> calculate absolute coordinate
	          #tempNextCmdIn.circleCenterPoint.x := #tempCurrentPoint.x + #nextCommandIn.cmdParameters.circleParameters.auxPoint[1];
	          #tempNextCmdIn.circleCenterPoint.y := #tempCurrentPoint.y + #nextCommandIn.cmdParameters.circleParameters.auxPoint[2];
	          #tempNextCmdIn.circleCenterPoint.z := #tempCurrentPoint.z + #nextCommandIn.cmdParameters.circleParameters.auxPoint[3];
	        END_IF;
	        IF (#tempNextCmdIn.circleMode = "CM_CENTER") THEN
	          // "Third" coordinate is ignored by system - also ignore here!
	          // Use start coordinate of circle instead
	          IF (#pathPlane = "CP_XZ") THEN
	            #tempNextCmdIn.circleCenterPoint.y := #tempCurrentPoint.y;
	          ELSIF (#pathPlane = "CP_YZ") THEN
	            #tempNextCmdIn.circleCenterPoint.x := #tempCurrentPoint.x;
	          ELSIF (#pathPlane = "CP_XY") THEN
	            #tempNextCmdIn.circleCenterPoint.z := #tempCurrentPoint.z;
	          END_IF;
	          
	          // Calculte correct circle end point - parameter not mandatory (and therefore probably not correct)
	          #tempRetValue := "LKinCtrl_CalcCircEndPointWithGivenCenterAndAngle"(circleStartPoint := #tempCurrentPoint,
	                                                                              circleCenterPoint := #tempNextCmdIn.circleCenterPoint,
	                                                                              pathPlane := #pathPlane,
	                                                                              pathChoice := #tempNextCmdIn.pathChoice,
	                                                                              angle := #tempNextCmdIn.circleAngle,
	                                                                              endPoint => #tempNextCmdIn.endPoint); // absolute coordinate
	          
	          IF (#tempRetValue <> 0) THEN
	            #LKinCtrl_OffsetContour.returnValue := #tempRetValue;
	            #LKinCtrl_OffsetContour."region" := #COFF_REGION_TYPE_PRE_CALC;
	            #LKinCtrl_OffsetContour.subBlockNumber := 35053;
	            #LKinCtrl_OffsetContour.internalNumber := 204;
	            RETURN;
	          END_IF;
	        END_IF;
	        
	      ELSE
	        #LKinCtrl_OffsetContour.returnValue := #ERR_COFF_INVALID_CIRCLE_MODE; // Invalid circle mode
	        #LKinCtrl_OffsetContour."region" := #COFF_REGION_TYPE_PLAUSIBILITY_NEXT_CMD;
	        RETURN;
	      END_IF;
	      
	      // Set command type to absolute
	      #tempNextCmdOut.cmdType := "LKINCTRL_MC_MOVECIRCULARABS";
	    ELSE
	      #LKinCtrl_OffsetContour.returnValue := #ERR_COFF_INVALID_COMMAND_TYPE; // Invalid command type
	      #LKinCtrl_OffsetContour."region" := #COFF_REGION_TYPE_PLAUSIBILITY_NEXT_CMD;
	      #LKinCtrl_OffsetContour.internalNumber := 205;
	      RETURN;
	    END_IF;
	    
	    // Write to output data - modifications done later
	    #tempNextCmdOut.circleMode := #tempNextCmdIn.circleMode;
	    #tempNextCmdOut.endPoint := #tempNextCmdIn.endPoint;
	    #tempNextCmdOut.circleIntermediatePoint := #tempNextCmdIn.circleIntermediatePoint;
	    #tempNextCmdOut.circleCenterPoint := #tempNextCmdIn.circleCenterPoint;
	    #tempNextCmdOut.transitionParameter1 := #tempNextCmdIn.transitionParameter1;
	    #tempNextCmdOut.circleAngle := #tempNextCmdIn.circleAngle;
	    
	    // Next but one command - important!
	    #tempNextButOneCmdIn.transitionParameter1 := #nextButOneCommandIn.cmdParameters.transitionParameters[1];
	    #tempNextButOneCmdOut.transitionParameter1 := #tempNextButOneCmdIn.transitionParameter1;
	  END_IF;
	END_REGION
	
	// Tool radius compensation
	REGION TOOL_RADIUS_COMPENSATION
	  // Copy important source variables into temporary variables
	  
	  IF (#tempToolRadiusComp) THEN
	    
	    REGION Copy data
	      // ############# C O P Y   D A T A #############
	      // #################################### 
	      
	      // Next but one command
	      //nextButOneCommandOut.transitionParameter := nextButOneCommandIn.cmdParameters.transitionParameters;
	      
	      // Next but one command
	      // --------------------------
	      #tempNextButOneCmdIn.cmdType := #nextButOneCommandIn.cmdType;
	      // Write to output data - modifications done later
	      #tempNextButOneCmdOut.cmdType := #tempNextButOneCmdIn.cmdType;
	      
	      
	      #tempNextButOneCmdIn.bufferMode := #nextButOneCommandIn.cmdParameters.bufferMode;
	      
	      // End point is defined
	      IF (#tempNextButOneCmdIn.cmdType = "LKINCTRL_MC_MOVELINEARABS") THEN
	        // Absolute coordinates
	        #tempNextButOneCmdIn.endPoint := "LKinCtrl_CartesianCoordTo3DPoint"(#nextButOneCommandIn.cmdCoordinates.cartesianPosition);
	        
	      ELSIF (#tempNextButOneCmdIn.cmdType = "LKINCTRL_MC_MOVELINEARREL") THEN
	        // Relative coordinates -> calculate absolute coordinate
	        #tempNextButOneCmdIn.endPoint := "LKinCtrl_VecAdd"(vIn1 := #tempNextCmdIn.endPoint,
	                                                           vIn2 := "LKinCtrl_CartesianCoordTo3DPoint"(#nextButOneCommandIn.cmdCoordinates.cartesianPosition));
	        
	        // Set command type to absolute
	        #tempNextButOneCmdOut.cmdType := "LKINCTRL_MC_MOVELINEARABS";
	        
	      ELSIF ((#tempNextButOneCmdIn.cmdType = "LKINCTRL_MC_MOVECIRCULARABS") OR
	        (#tempNextButOneCmdIn.cmdType = "LKINCTRL_MC_MOVECIRCULARREL"))
	      THEN
	        #tempNextButOneCmdIn.circleMode := #nextButOneCommandIn.cmdParameters.circleParameters.circMode;
	        #tempNextButOneCmdIn.pathChoice := #nextButOneCommandIn.cmdParameters.circleParameters.pathChoice;
	        
	        // Check for invalid path choice
	        IF ((#tempNextButOneCmdIn.pathChoice < "PC_POSITIVE") OR
	          (#tempNextButOneCmdIn.pathChoice > "PC_NEGATIVE"))
	        THEN
	          #LKinCtrl_OffsetContour.returnValue := #ERR_COFF_INVALID_PATH_CHOICE_OF_CIRCULAR_CMD; // Invalid path plane of a circular command
	          #LKinCtrl_OffsetContour."region" := #COFF_REGION_TYPE_PLAUSIBILITY_NEXT_BUT_ONE_CMD;
	          #LKinCtrl_OffsetContour.internalNumber := 210;
	          RETURN;
	        END_IF;
	        
	        #tempNextButOneCmdIn.circlePlane := #nextButOneCommandIn.cmdParameters.circleParameters.circlePlane;
	        
	        IF ((#tempNextButOneCmdIn.circleMode = "CM_BORDER") OR
	          (#tempNextButOneCmdIn.circleMode = "CM_RADIUS"))
	        THEN
	          
	          // End point is defined
	          IF (#tempNextButOneCmdIn.cmdType = "LKINCTRL_MC_MOVECIRCULARABS") THEN
	            // Absolute coordinates
	            #tempNextButOneCmdIn.endPoint := "LKinCtrl_CartesianCoordTo3DPoint"(#nextButOneCommandIn.cmdCoordinates.cartesianPosition);
	          ELSE
	            // Relative coordinates -> calculate absolute coordinate 
	            #tempNextButOneCmdIn.endPoint := "LKinCtrl_VecAdd"(vIn1 := #tempNextCmdIn.endPoint,
	                                                               vIn2 := "LKinCtrl_CartesianCoordTo3DPoint"(#nextButOneCommandIn.cmdCoordinates.cartesianPosition));
	          END_IF;
	          
	          IF (#tempNextButOneCmdIn.circleMode = "CM_BORDER") THEN
	            IF (#tempNextButOneCmdIn.cmdType = "LKINCTRL_MC_MOVECIRCULARABS") THEN
	              // Absolute coordinates
	              #tempNextButOneCmdIn.circleIntermediatePoint.x := #nextButOneCommandIn.cmdParameters.circleParameters.auxPoint[1];
	              #tempNextButOneCmdIn.circleIntermediatePoint.y := #nextButOneCommandIn.cmdParameters.circleParameters.auxPoint[2];
	              #tempNextButOneCmdIn.circleIntermediatePoint.z := #nextButOneCommandIn.cmdParameters.circleParameters.auxPoint[3];
	            ELSE
	              // Relative coordinates -> calculate absolute coordinate
	              #tempNextButOneCmdIn.circleIntermediatePoint.x := #tempNextCmdIn.endPoint.x + #nextButOneCommandIn.cmdParameters.circleParameters.auxPoint[1];
	              #tempNextButOneCmdIn.circleIntermediatePoint.y := #tempNextCmdIn.endPoint.y + #nextButOneCommandIn.cmdParameters.circleParameters.auxPoint[2];
	              #tempNextButOneCmdIn.circleIntermediatePoint.z := #tempNextCmdIn.endPoint.z + #nextButOneCommandIn.cmdParameters.circleParameters.auxPoint[3];
	            END_IF;
	          END_IF;
	          
	          IF (#tempNextButOneCmdIn.circleMode = "CM_RADIUS") THEN
	            #tempNextButOneCmdIn.circleRadius := #nextButOneCommandIn.cmdParameters.circleParameters.radius;
	            
	            // "Third" coordinate is ignored by system - also ignore here!
	            // Use start coordinate of circle instead
	            IF (#pathPlane = "CP_XZ") THEN
	              #tempNextButOneCmdIn.endPoint.y := #tempNextCmdIn.endPoint.y;
	            ELSIF (#pathPlane = "CP_YZ") THEN
	              #tempNextButOneCmdIn.endPoint.x := #tempNextCmdIn.endPoint.x;
	            ELSIF (#pathPlane = "CP_XY") THEN
	              #tempNextButOneCmdIn.endPoint.z := #tempNextCmdIn.endPoint.z;
	            END_IF;
	            
	          END_IF;
	          
	        ELSIF (#tempNextButOneCmdIn.circleMode = "CM_CENTER") THEN
	          #tempNextButOneCmdIn.circleAngle := #nextButOneCommandIn.cmdParameters.circleParameters.arc;
	          
	          IF (#tempNextButOneCmdIn.cmdType = "LKINCTRL_MC_MOVECIRCULARABS") THEN
	            // Absolute coordinates
	            #tempNextButOneCmdIn.circleCenterPoint.x := #nextButOneCommandIn.cmdParameters.circleParameters.auxPoint[1];
	            #tempNextButOneCmdIn.circleCenterPoint.y := #nextButOneCommandIn.cmdParameters.circleParameters.auxPoint[2];
	            #tempNextButOneCmdIn.circleCenterPoint.z := #nextButOneCommandIn.cmdParameters.circleParameters.auxPoint[3];
	          ELSE
	            // Relative coordinates -> calculate absolute coordinate
	            #tempNextButOneCmdIn.circleCenterPoint.x := #tempNextCmdIn.endPoint.x + #nextButOneCommandIn.cmdParameters.circleParameters.auxPoint[1];
	            #tempNextButOneCmdIn.circleCenterPoint.y := #tempNextCmdIn.endPoint.y + #nextButOneCommandIn.cmdParameters.circleParameters.auxPoint[2];
	            #tempNextButOneCmdIn.circleCenterPoint.z := #tempNextCmdIn.endPoint.z + #nextButOneCommandIn.cmdParameters.circleParameters.auxPoint[3];
	          END_IF;
	          
	          // "Third" coordinate is ignored by system - also ignore here!
	          // Use start coordinate of circle instead
	          IF (#pathPlane = "CP_XZ") THEN
	            #tempNextButOneCmdIn.circleCenterPoint.y := #tempNextCmdIn.endPoint.y;
	          ELSIF (#pathPlane = "CP_YZ") THEN
	            #tempNextButOneCmdIn.circleCenterPoint.x := #tempNextCmdIn.endPoint.x;
	          ELSIF (#pathPlane = "CP_XY") THEN
	            #tempNextButOneCmdIn.circleCenterPoint.z := #tempNextCmdIn.endPoint.z;
	          END_IF;
	          
	        ELSE
	          #LKinCtrl_OffsetContour.returnValue := #ERR_COFF_INVALID_CIRCLE_MODE; // Invalid circle mode
	          #LKinCtrl_OffsetContour."region" := #COFF_REGION_TYPE_PLAUSIBILITY_NEXT_BUT_ONE_CMD;
	          #LKinCtrl_OffsetContour.internalNumber := 211;
	          RETURN;
	        END_IF;
	        
	        // Set command type to absolute
	        #tempNextButOneCmdOut.cmdType := "LKINCTRL_MC_MOVECIRCULARABS";
	        
	      ELSIF (#tempNextButOneCmdIn.cmdType = -1) THEN
	        ;
	      ELSE
	        #LKinCtrl_OffsetContour.returnValue := #ERR_COFF_INVALID_COMMAND_TYPE; // Invalid command type
	        #LKinCtrl_OffsetContour."region" := #COFF_REGION_TYPE_PLAUSIBILITY_NEXT_BUT_ONE_CMD;
	        #LKinCtrl_OffsetContour.internalNumber := 212;
	        RETURN;
	      END_IF;
	      
	      // Write to output data - modifications done later
	      #tempNextButOneCmdOut.circleMode := #tempNextButOneCmdIn.circleMode;
	      #tempNextButOneCmdOut.endPoint := #tempNextButOneCmdIn.endPoint;
	      #tempNextButOneCmdOut.circleIntermediatePoint := #tempNextButOneCmdIn.circleIntermediatePoint;
	      #tempNextButOneCmdOut.circleCenterPoint := #tempNextButOneCmdIn.circleCenterPoint;
	      
	      
	    END_REGION
	    
	    REGION Next command LINEAR
	      
	      // ############# N E X T   C M D  -  L I N E A R #############
	      // ##############################################
	      IF (#tempNextCmdOut.cmdType = "LKINCTRL_MC_MOVELINEARABS") THEN
	        IF (#boCmdInPathPlane) THEN
	          // ########## 1st linear command point 1 to point 2 ##########
	          // Calculate tangential and orthogonal unit vector of direction
	          #tempRetValue := "LKinCtrl_CalcLineTangOrthPathPlane"(pathPlane := #pathPlane,
	                                                                compDirection := #compensationDirection,
	                                                                vInFirst := #tempNextCmdIn.endPoint,
	                                                                vInSecond := #tempCurrentPoint,
	                                                                vUnitTangentialPathPlane => #tempNextCmdOut.tangentialUnitVecEnd,
	                                                                vUnitOrthogonalPathPlane => #tempNextCmdOut.orthogonalUnitVecEnd);
	          
	          IF (#tempRetValue <> 0) THEN
	            #LKinCtrl_OffsetContour.returnValue := #tempRetValue;
	            #LKinCtrl_OffsetContour."region" := #COFF_REGION_TYPE_RAD_COMP_NEXT_CMD_LIN;
	            #LKinCtrl_OffsetContour.subBlockNumber := 35055;
	            #LKinCtrl_OffsetContour.internalNumber := 301;
	            RETURN;
	          END_IF;
	          
	          // Scale othogonal vector with tool radius to get orthogonal shift
	          #tempNextCmdOut.orthogonalShiftEnd := "LKinCtrl_VecScale"(vIn := #tempNextCmdOut.orthogonalUnitVecEnd,
	                                                                    factor := #toolRadius);
	          
	          // Scale tangential vector with tool radius to get tangential shift
	          #tempNextCmdOut.tangentiaShiftEnd := "LKinCtrl_VecScale"(vIn := #tempNextCmdOut.tangentialUnitVecEnd,
	                                                                   factor := #toolRadius);
	          
	          // Calculate orthogonal shifted next target coordinate 
	          #tempNextCmdOut.endPointOrthShifted := "LKinCtrl_VecAdd"(vIn1 := #tempNextCmdIn.endPoint,
	                                                                   vIn2 := #tempNextCmdOut.orthogonalShiftEnd);
	          
	          // Calculate orthogonal and tangential shifted next target coordinate
	          #tempNextCmdOut.endPointOrthTangShifted := "LKinCtrl_VecAdd"(vIn1 := #tempNextCmdOut.endPointOrthShifted,
	                                                                       vIn2 := #tempNextCmdOut.tangentiaShiftEnd);
	          
	          #tempNextCmdOut.endPoint := #tempNextCmdOut.endPointOrthShifted;
	          
	          // ############# N E X T   B U T   O N E   C M D  -  L I N E A R #############
	          IF (#tempNextButOneCmdOut.cmdType = "LKINCTRL_MC_MOVELINEARABS") THEN
	            REGION Next but one command LINEAR
	              // 2nd linear command point 2 to point 3
	              // Calculate tangential and orthogonal unit vector of direction
	              #tempRetValue := "LKinCtrl_CalcLineTangOrthPathPlane"(pathPlane := #pathPlane,
	                                                                    compDirection := #compensationDirection,
	                                                                    vInFirst := #tempNextButOneCmdIn.endPoint,
	                                                                    vInSecond := #tempNextCmdIn.endPoint,
	                                                                    vUnitTangentialPathPlane => #tempNextButOneCmdOut.tangentialUnitVecStart,
	                                                                    vUnitOrthogonalPathPlane => #tempNextButOneCmdOut.orthogonalUnitVecStart);
	              
	              IF (#tempRetValue <> 0) THEN
	                #LKinCtrl_OffsetContour.returnValue := #tempRetValue;
	                #LKinCtrl_OffsetContour."region" := #COFF_REGION_TYPE_RAD_COMP_LIN_LIN;
	                #LKinCtrl_OffsetContour.subBlockNumber := 35055;
	                #LKinCtrl_OffsetContour.internalNumber := 302;
	                RETURN;
	              END_IF;
	              
	              // Scale othogonal vector with tool radius to get orthogonal shift
	              #tempNextButOneCmdOut.orthogonalShiftStart := "LKinCtrl_VecScale"(vIn := #tempNextButOneCmdOut.orthogonalUnitVecStart,
	                                                                                factor := #toolRadius);
	              
	              #tempNextButOneCmdOut.tangentiaShiftStart := "LKinCtrl_VecScale"(vIn := #tempNextButOneCmdOut.tangentialUnitVecStart,
	                                                                               factor := #toolRadius);
	              
	              // Calculate orthogonal shifted next target coordinate 
	              #tempNextButOneCmdOut.startPointOrthShifted := "LKinCtrl_VecAdd"(vIn1 := #tempNextCmdIn.endPoint,
	                                                                               vIn2 := #tempNextButOneCmdOut.orthogonalShiftStart);
	              
	              // Calculate orthogonal and tangential shifted next target coordinate
	              #tempNextButOneCmdOut.startPointOrthTangShifted := "LKinCtrl_VecAdd"(vIn1 := #tempNextButOneCmdOut.startPointOrthShifted,
	                                                                                   vIn2 := #tempNextButOneCmdOut.tangentiaShiftStart);
	              
	              // Check if 1st and 2nd linear command are located in exactly the same direction (tangential vector) - then orhtogonal shifted end point of next command is the solution!
	              // No intersection point, lines intersect completely!
	              #tempDistance1 := ("LKinCtrl_VecAbs"("LKinCtrl_VecSub"(vIn1 := #tempNextCmdOut.tangentialUnitVecEnd, vIn2 := #tempNextButOneCmdOut.tangentialUnitVecStart)));
	              
	              // Check for zero vector
	              #tempDistance2 := ("LKinCtrl_VecAbs"(#tempNextButOneCmdOut.tangentialUnitVecStart));
	              
	              IF ((#tempDistance1 > #COFF_TOLERANCE) AND (#tempDistance2 > 0.0)) THEN
	                // ########## Intersection point of 1st and 2nd linear command ##########
	                #tempRetValue := "LKinCtrl_CalcLineLineIntersectionPoint"(startPointFirstLine := #tempNextCmdOut.endPointOrthShifted,
	                                                                          endPointFirstLine := #tempNextCmdOut.endPointOrthTangShifted,
	                                                                          startPointSecondLine := #tempNextButOneCmdOut.startPointOrthShifted,
	                                                                          endPointSecondLine := #tempNextButOneCmdOut.startPointOrthTangShifted,
	                                                                          intersectionPointA => #tempPa,
	                                                                          intersectionPointB => #tempPb,
	                                                                          muA => #tempMuA,
	                                                                          muB => #tempMuB);
	                
	                IF (#tempRetValue <> 0) THEN
	                  #LKinCtrl_OffsetContour.returnValue := #tempRetValue;
	                  #LKinCtrl_OffsetContour."region" := #COFF_REGION_TYPE_RAD_COMP_LIN_LIN;
	                  #LKinCtrl_OffsetContour.subBlockNumber := 35060;
	                  #LKinCtrl_OffsetContour.internalNumber := 303;
	                  RETURN;
	                END_IF;
	                #tempNextCmdOut.endPoint := #tempPa;
	              ELSE
	                #tempNextCmdOut.endPoint := #tempNextCmdOut.endPointOrthShifted;
	              END_IF;
	              
	              // Check blending length
	              IF ((#tempNextButOneCmdIn.transitionParameter1 < 0.0) OR
	                // V01.01.02 AW 2020-10-13 - avoid inner / outer corner check if 1st and 2nd linear command are located in exactly the same direction
	                (#tempDistance1 < #COFF_TOLERANCE))
	              THEN
	                ; // Maximum blending length used - automatic algorithm, nothing to change here
	                // OR nothing to do - straight line
	              ELSE
	                // Distinguish between inner and outer corner
	                #tempRetValue := "LKinCtrl_CheckInnerOuterCorner"(vInFirst := #tempNextCmdOut.tangentialUnitVecEnd,
	                                                                  vInSecond := #tempNextButOneCmdOut.tangentialUnitVecStart,
	                                                                  pathPlane := #pathPlane,
	                                                                  direction := #compensationDirection,
	                                                                  cornerType => #tempCornerType);
	                
	                IF (#tempRetValue <> 0) THEN
	                  #LKinCtrl_OffsetContour.returnValue := #tempRetValue;
	                  #LKinCtrl_OffsetContour."region" := #COFF_REGION_TYPE_RAD_COMP_LIN_LIN;
	                  #LKinCtrl_OffsetContour.subBlockNumber := 35051;
	                  #LKinCtrl_OffsetContour.internalNumber := 304;
	                  RETURN;
	                END_IF;
	                
	                IF (#tempCornerType = "LKINCTRL_OUTER_CORNER") THEN
	                  IF (#tempNextButOneCmdIn.transitionParameter1 > #COFF_TRANSITION_TOLERANCE) THEN
	                    
	                    // Output next but one coordinates - in case it's the last one
	                    #tempNextButOneCmdOut.endPoint := "LKinCtrl_VecAdd"(vIn1 := #tempNextButOneCmdIn.endPoint,
	                                                                        vIn2 := #tempNextButOneCmdOut.orthogonalShiftStart);
	                    
	                    
	                    // Modify transition with blending distance - next but one command !
	                    #tempNextButOneCmdOut.transitionParameter1 += #toolRadius;
	                    
	                  ELSE
	                    // Use shortened end point
	                    #tempNextCmdOut.endPoint := #tempNextCmdOut.endPointOrthShifted;
	                    
	                    // Additional command
	                    // Intermediate command necessary (circle defined by intermediate position)
	                    "LKinCtrl_CalcCircleIntermediatePos"(initialEndPoint := #tempNextCmdIn.endPoint,
	                                                         newEndPoint := #tempPa,
	                                                         toolRadius := #toolRadius,
	                                                         circIntermediatePoint => #tempIntermediateCmdOut.circleIntermediatePoint);
	                    
	                    
	                    #tempIntermediateCmdOut.cmdType := "LKINCTRL_MC_MOVECIRCULARABS";
	                    
	                    #tempIntermediateCmdOut.endPoint := #tempNextButOneCmdOut.startPointOrthShifted;
	                    
	                    // Definition via intermediate point and endpoint
	                    #tempIntermediateCmdOut.circleMode := "CM_BORDER";
	                    
	                  END_IF;
	                ELSE // Inner corner
	                  ;
	                END_IF;
	              END_IF;
	            END_REGION
	            // #############  N E X T   B U T   O N E   C M D   -  C I R C U L A R #############
	          ELSIF (#tempNextButOneCmdOut.cmdType = "LKINCTRL_MC_MOVECIRCULARABS") THEN
	            REGION Next but one command CIRCULAR
	              // Use radius-compensated point (linear end point)
	              //nextCommandOut.cmdCoordinates.cartesianPosition := #tempNew2ndPoint;
	              
	              // Distinguish between different circular modes
	              IF (#tempNextButOneCmdIn.circleMode = "CM_BORDER") THEN
	                
	                // ------------ Via an intermediate point and the end point ("CircMode" = 0) ------------
	                
	                // Caluclate center point of circle with given start point, end point and intermediate point
	                #tempRetValue := "LKinCtrl_CalcCircCenterByIntermediatePointAndEndPoint"(circleStartPoint := #tempNextCmdIn.endPoint,
	                                                                                         circleEndPoint := #tempNextButOneCmdIn.endPoint,
	                                                                                         circleIntermediatePoint := #tempNextButOneCmdIn.circleIntermediatePoint,
	                                                                                         pathPlane := #pathPlane,
	                                                                                         circleCenterPoint => #tempNextButOneCmdIn.circleCenterPoint);
	                
	                IF (#tempRetValue <> 0) THEN
	                  #LKinCtrl_OffsetContour.returnValue := #tempRetValue;
	                  #LKinCtrl_OffsetContour."region" := #COFF_REGION_TYPE_RAD_COMP_LIN_CIRC;
	                  #LKinCtrl_OffsetContour.subBlockNumber := 35057;
	                  #LKinCtrl_OffsetContour.internalNumber := 330;
	                  RETURN;
	                END_IF;
	                
	                // Calculate path choice
	                #tempRetValue := "LKinCtrl_CalcCircPathChoiceByIntermediatePointAndEndPoint"(circleStartPoint := #tempNextCmdIn.endPoint,
	                                                                                             circleEndPoint := #tempNextButOneCmdIn.endPoint,
	                                                                                             circleintermediatePoint := #tempNextButOneCmdIn.circleIntermediatePoint,
	                                                                                             pathPlane := #pathPlane,
	                                                                                             pathChoice => #tempNextButOneCmdIn.pathChoice);
	                
	                
	                IF (#tempRetValue <> 0) THEN
	                  #LKinCtrl_OffsetContour.returnValue := #tempRetValue;
	                  #LKinCtrl_OffsetContour."region" := #COFF_REGION_TYPE_RAD_COMP_LIN_CIRC;
	                  #LKinCtrl_OffsetContour.subBlockNumber := 35058;
	                  #LKinCtrl_OffsetContour.internalNumber := 331;
	                  RETURN;
	                END_IF;
	                
	              ELSIF (#tempNextButOneCmdIn.circleMode = "CM_CENTER") THEN
	                // ------------ Via the circle center and the angle in a main plane ("CircMode" = 1) ------------
	                // "Third" coordinate is ignored by system - also ignore here!
	                
	                // Calculte correct circle end point - parameter not mandatory (and therefore probably not correct)
	                #tempRetValue := "LKinCtrl_CalcCircEndPointWithGivenCenterAndAngle"(circleStartPoint := #tempNextCmdIn.endPoint,
	                                                                                    circleCenterPoint := #tempNextButOneCmdIn.circleCenterPoint,
	                                                                                    pathPlane := #pathPlane,
	                                                                                    pathChoice := #tempNextButOneCmdIn.pathChoice,
	                                                                                    angle := #tempNextButOneCmdIn.circleAngle,
	                                                                                    endPoint => #tempNextButOneCmdIn.endPoint);
	                
	                
	                
	                
	                IF (#tempRetValue <> 0) THEN
	                  #LKinCtrl_OffsetContour.returnValue := #tempRetValue;
	                  #LKinCtrl_OffsetContour."region" := #COFF_REGION_TYPE_RAD_COMP_CIRC_CIRC;
	                  #LKinCtrl_OffsetContour.subBlockNumber := 35053;
	                  #LKinCtrl_OffsetContour.internalNumber := 332;
	                  RETURN;
	                END_IF;
	                
	              ELSIF (#tempNextButOneCmdIn.circleMode = "CM_RADIUS") THEN
	                
	                // Calculate circle center point by given start / end point and radius and path choice
	                #tempRetValue := "LKinCtrl_CalcCircCenterByRadiusAndEndPoint"(circleStartPoint := #tempNextCmdIn.endPoint,
	                                                                              circleEndPoint := #tempNextButOneCmdIn.endPoint,
	                                                                              pathPlane := #pathPlane,
	                                                                              circleRadius := #tempNextButOneCmdIn.circleRadius,
	                                                                              pathChoice := #tempNextButOneCmdIn.pathChoice,
	                                                                              circCenterPoint => #tempNextButOneCmdIn.circleCenterPoint);
	                
	                IF (#tempRetValue <> 0) THEN
	                  #LKinCtrl_OffsetContour.returnValue := #tempRetValue;
	                  #LKinCtrl_OffsetContour."region" := #COFF_REGION_TYPE_RAD_COMP_LIN_CIRC;
	                  #LKinCtrl_OffsetContour.subBlockNumber := 35052;
	                  #LKinCtrl_OffsetContour.internalNumber := 333;
	                  RETURN;
	                END_IF;
	                
	                
	                
	              END_IF;
	              
	              // Calculate end coordinate of "next" linear command
	              // Calculate orthogonal and tangential vector for next but one circular commamnd
	              #tempRetValue := "LKinCtrl_CalcCircTangOrthPathPlane"(circlePoint := #tempNextCmdIn.endPoint,
	                                                                    circleCenterPoint := #tempNextButOneCmdIn.circleCenterPoint,
	                                                                    pathPlane := #pathPlane,
	                                                                    compDirection := #compensationDirection,
	                                                                    pathChoice := #tempNextButOneCmdIn.pathChoice,
	                                                                    vUnitTangentialPathPlane => #tempNextButOneCmdOut.tangentialUnitVecStart,
	                                                                    vUnitOrthogonalPathPlane => #tempNextButOneCmdOut.orthogonalUnitVecStart);
	              
	              IF (#tempRetValue <> 0) THEN
	                #LKinCtrl_OffsetContour.returnValue := #tempRetValue;
	                #LKinCtrl_OffsetContour."region" := #COFF_REGION_TYPE_RAD_COMP_LIN_CIRC;
	                #LKinCtrl_OffsetContour.subBlockNumber := 35056;
	                #LKinCtrl_OffsetContour.internalNumber := 334;
	                RETURN;
	              END_IF;
	              
	              
	              // Scale othogonal vector with tool radius to get orthogonal shift
	              #tempNextButOneCmdOut.orthogonalShiftStart := "LKinCtrl_VecScale"(vIn := #tempNextButOneCmdOut.orthogonalUnitVecStart,
	                                                                                factor := #toolRadius);
	              
	              #tempNextButOneCmdOut.startPointOrthShifted := "LKinCtrl_VecAdd"(vIn1 := #tempNextCmdIn.endPoint,
	                                                                               vIn2 := #tempNextButOneCmdOut.orthogonalShiftStart);
	              
	              // Calculate radius of circle
	              #tempNextCmdOut.circleRadius := "LKinCtrl_VecAbs"("LKinCtrl_VecSub"(vIn1 := #tempNextButOneCmdOut.startPointOrthShifted,
	                                                                                                                                    vIn2 := #tempNextButOneCmdIn.circleCenterPoint));
	              
	              
	              // ########## Intersection point of 1st linear and 2nd circular command  ##########
	              // V01.02.01 - bugfix linear start point
	              #tempRetValue := "LKinCtrl_CalcLineCircleIntersectionPoint"(startPointLine := #tempCurrentPointRadComp,//tempNextCmdOut.endPointOrthShifted,
	                                                                          endPointLine := #tempNextCmdOut.endPointOrthTangShifted,
	                                                                          circleCenter := #tempNextButOneCmdIn.circleCenterPoint,
	                                                                          circleRadius := #tempNextCmdOut.circleRadius,
	                                                                          intersectionPointA => #tempPa,
	                                                                          intersectionPointB => #tempPb);
	              
	              IF (#tempRetValue <> 0) THEN
	                #LKinCtrl_OffsetContour.returnValue := #tempRetValue;
	                #LKinCtrl_OffsetContour."region" := #COFF_REGION_TYPE_RAD_COMP_LIN_CIRC;
	                #LKinCtrl_OffsetContour.subBlockNumber := 35061;
	                #LKinCtrl_OffsetContour.internalNumber := 335;
	                RETURN;
	              END_IF;
	              
	              
	              // Two intersection points, use the one which is closer to the circle start point
	              #tempDistance1 := "LKinCtrl_VecAbs"("LKinCtrl_VecSub"(vIn1 := #tempNextCmdOut.endPointOrthShifted, vIn2 := #tempPa));
	              #tempDistance2 := "LKinCtrl_VecAbs"("LKinCtrl_VecSub"(vIn1 := #tempNextCmdOut.endPointOrthShifted, vIn2 := #tempPb));
	              
	              IF (#tempDistance1 < #tempDistance2) THEN
	                #tempNextCmdOut.endPoint := #tempPa;
	              ELSE
	                #tempNextCmdOut.endPoint := #tempPb;
	              END_IF;
	              
	            END_REGION
	            // ############# N E X T   B U T   O N E   C M D  -  N O N E #############
	          ELSE
	            REGION Next but one command NONE
	              // V01.01.02 AW 2020-10-13
	              // Check if current end point is in opposite direction, e.g. small command length with big tool radius etc.
	              // Avoid reversal movement
	              
	              // Calculate difference vector of uncompensated current and next end point
	              #tempDirectionUncompensatedVec := "LKinCtrl_VecSub"(vIn1 := #tempCurrentPoint, vIn2 := #tempNextCmdIn.endPoint);
	              #tempDirectionUncompensatedUnitVec := "LKinCtrl_VecUnit"(#tempDirectionUncompensatedVec);
	              
	              // Calculate difference vector of compensated current and next end point
	              #tempDirectionCompensatedVec := "LKinCtrl_VecSub"(vIn1 := #tempCurrentPointRadComp, vIn2 := #tempNextCmdOut.endPoint);
	              #tempDirectionCompensatedUnitVec := "LKinCtrl_VecUnit"(#tempDirectionCompensatedVec);
	              
	              // Calculate length between current compensated and next compensated end point
	              #tempLengthCompensatedPointDifferenceVec := "LKinCtrl_VecAbs"(#tempDirectionCompensatedVec);
	              
	              // Check if vectors are parallel 
	              IF (((ABS(#tempDirectionUncompensatedUnitVec.x) - ABS(#tempDirectionCompensatedUnitVec.x)) < #COFF_TOLERANCE) AND
	                ((ABS(#tempDirectionUncompensatedUnitVec.y) - ABS(#tempDirectionCompensatedUnitVec.y)) < #COFF_TOLERANCE) AND
	                ((ABS(#tempDirectionUncompensatedUnitVec.z) - ABS(#tempDirectionCompensatedUnitVec.z)) < #COFF_TOLERANCE))
	              THEN
	                // Opposite direction?
	                IF ((ABS(#tempDirectionUncompensatedUnitVec.x + #tempDirectionCompensatedUnitVec.x) < #COFF_TOLERANCE) AND
	                  (ABS(#tempDirectionUncompensatedUnitVec.y + #tempDirectionCompensatedUnitVec.y) < #COFF_TOLERANCE) AND
	                  (ABS(#tempDirectionUncompensatedUnitVec.z + #tempDirectionCompensatedUnitVec.z) < #COFF_TOLERANCE))
	                THEN
	                  // Throw error
	                  #LKinCtrl_OffsetContour.returnValue := #ERR_COFF_LINEAR_CMD_AND_TOOL_RADIUS_LEAD_TO_REVERSAL;
	                  #LKinCtrl_OffsetContour."region" := #COFF_REGION_TYPE_RAD_COMP_LIN_NONE;
	                  #LKinCtrl_OffsetContour.subBlockNumber := 0;
	                  #LKinCtrl_OffsetContour.internalNumber := 336;
	                  RETURN;
	                  
	                  // // Possible solution - NOT used!
	                  // // Use tangential and orthogonal shift
	                  // // Scale tangential vector with point difference (compensated points) to get tangential shift
	                  // #tempNextCmdOut.tangentiaShiftEnd := "LKinCtrl_VecScale"(vIn := #tempNextCmdOut.tangentialUnitVecEnd,
	                  //                                                          factor := #tempLengthCompensatedPointDifferenceVec);
	                  
	                  // // Re-calculate orthogonal and (new) tangential shifted next target coordinate
	                  // // next command end point will be equal to last command end point --> no reversal
	                  // #tempNextCmdOut.endPointOrthTangShifted := "LKinCtrl_VecAdd"(vIn1 := #tempNextCmdOut.endPointOrthShifted,
	                  //                                                              vIn2 := #tempNextCmdOut.tangentiaShiftEnd);
	                  
	                  // // Use tangential and orthogonal shift - assign new value
	                  // #tempNextCmdOut.endPoint := #tempNextCmdOut.endPointOrthTangShifted;
	                  
	                ELSE
	                  // Same direction
	                  ;// Nothing to do
	                END_IF;
	              ELSE
	                // V01.01.03
	                ;// Nothing to do
	              END_IF;
	              
	            END_REGION
	          END_IF;
	          
	          REGION Additional plausibility check
	            #tempRetValue := "LKinCtrl_CalcAngleBetweenVectors"(point1 := #tempNextCmdOut.endPoint,
	                                                                point2 := #tempNextCmdIn.endPoint,
	                                                                intersectionPoint := #tempCurrentPoint,
	                                                                angle => #tempAngle);
	            
	            IF (#tempRetValue <> 0) THEN
	              #LKinCtrl_OffsetContour.returnValue := #tempRetValue;
	              #LKinCtrl_OffsetContour."region" := #COFF_REGION_TYPE_RAD_COMP_LIN_GEN;
	              #LKinCtrl_OffsetContour.subBlockNumber := 35059;
	              #LKinCtrl_OffsetContour.internalNumber := 340;
	              RETURN;
	            END_IF;
	            
	            IF (#tempAngle > #COFF_CIRC_REVERSAL_TOLERANCE_ANGLE)
	            THEN
	              #LKinCtrl_OffsetContour.returnValue := #ERR_COFF_NO_SOLUTION_FOR_GIVEN_LINEAR_CMD;
	              #LKinCtrl_OffsetContour."region" := #COFF_REGION_TYPE_RAD_COMP_LIN_GEN;
	              #LKinCtrl_OffsetContour.subBlockNumber := 0;
	              #LKinCtrl_OffsetContour.internalNumber := 341;
	              RETURN;
	            END_IF;
	            
	          END_REGION
	        ELSE
	          // Use radius compensated coordinates
	          CASE #pathPlane OF
	            "CP_XY":
	              #tempNextCmdOut.endPoint.x := #tempCurrentPointRadComp.x;
	              #tempNextCmdOut.endPoint.y := #tempCurrentPointRadComp.y;
	              #tempNextCmdOut.endPoint.z := #tempNextCmdOut.endPoint.z;
	              
	            "CP_XZ":
	              #tempNextCmdOut.endPoint.x := #tempCurrentPointRadComp.x;
	              #tempNextCmdOut.endPoint.y := #tempNextCmdOut.endPoint.y;
	              #tempNextCmdOut.endPoint.z := #tempCurrentPointRadComp.z;
	              
	            "CP_YZ":
	              #tempNextCmdOut.endPoint.x := #tempNextCmdOut.endPoint.x;
	              #tempNextCmdOut.endPoint.y := #tempCurrentPointRadComp.y;
	              #tempNextCmdOut.endPoint.z := #tempCurrentPointRadComp.z;
	          END_CASE;
	        END_IF;
	      END_IF;
	    END_REGION
	    
	    REGION Next command CIRCULAR
	      // ############# N E X T   C M D  -  C I R C U L A R #############
	      // ##############################################
	      IF (#tempNextCmdOut.cmdType = "LKINCTRL_MC_MOVECIRCULARABS") THEN
	        
	        // Distinguish between different circular modes
	        IF (#tempNextCmdIn.circleMode = "CM_BORDER") THEN
	          
	          // ------------ Via an intermediate point and the end point ("CircMode" = 0) ------------
	          // Caluclate center point of circle with given start point, end point and intermediate point
	          #tempRetValue := "LKinCtrl_CalcCircCenterByIntermediatePointAndEndPoint"(circleStartPoint := #tempCurrentPoint,
	                                                                                   circleEndPoint := #tempNextCmdIn.endPoint,
	                                                                                   circleIntermediatePoint := #tempNextCmdIn.circleIntermediatePoint,
	                                                                                   pathPlane := #pathPlane,
	                                                                                   circleCenterPoint => #tempNextCmdIn.circleCenterPoint);
	          
	          IF (#tempRetValue <> 0) THEN
	            #LKinCtrl_OffsetContour.returnValue := #tempRetValue;
	            #LKinCtrl_OffsetContour."region" := #COFF_REGION_TYPE_RAD_COMP_NEXT_CMD_CIRC;
	            #LKinCtrl_OffsetContour.subBlockNumber := 35057;
	            
	            #LKinCtrl_OffsetContour.internalNumber := 401;
	            RETURN;
	          END_IF;
	          
	          // Calculate path choice
	          #tempRetValue := "LKinCtrl_CalcCircPathChoiceByIntermediatePointAndEndPoint"(circleStartPoint := #tempCurrentPoint,
	                                                                                       circleEndPoint := #tempNextCmdIn.endPoint,
	                                                                                       circleintermediatePoint := #tempNextCmdIn.circleIntermediatePoint,
	                                                                                       pathPlane := #pathPlane,
	                                                                                       pathChoice => #tempNextCmdIn.pathChoice);
	          
	          IF (#tempRetValue <> 0) THEN
	            #LKinCtrl_OffsetContour.returnValue := #tempRetValue;
	            #LKinCtrl_OffsetContour."region" := #COFF_REGION_TYPE_RAD_COMP_NEXT_CMD_CIRC;
	            #LKinCtrl_OffsetContour.subBlockNumber := 35058;
	            #LKinCtrl_OffsetContour.internalNumber := 402;
	            RETURN;
	          END_IF;
	          
	        ELSIF (#tempNextCmdIn.circleMode = "CM_CENTER") THEN
	          // ------------ Via the circle center and the angle in a main plane ("CircMode" = 1) ------------
	          (* im oberen Teil!
	          // "Third" coordinate is ignored by system - also ignore here!
	          // Use start coordinate of circle instead
	          IF (#pathPlane = "CP_XZ") THEN
	            #tempNextCmdIn.circleCenterPoint.y := #tempCurrentPoint.y;
	          ELSIF (#pathPlane = "CP_YZ") THEN
	            #tempNextCmdIn.circleCenterPoint.x := #tempCurrentPoint.x;
	          ELSIF (#pathPlane = "CP_XY") THEN
	            #tempNextCmdIn.circleCenterPoint.z := #tempCurrentPoint.z;
	          END_IF;*)
	          ;
	          
	        ELSIF (#tempNextCmdIn.circleMode = "CM_RADIUS") THEN
	          // ------------ Via the circle radius and the end point in a main plane ("CircMode" = 2) ------------
	          // Calculate circle center point by given start / end point and radius and path choice
	          #tempRetValue := "LKinCtrl_CalcCircCenterByRadiusAndEndPoint"(circleStartPoint := #tempCurrentPoint,
	                                                                        circleEndPoint := #tempNextCmdIn.endPoint,
	                                                                        pathPlane := #pathPlane,
	                                                                        circleRadius := #tempNextCmdIn.circleRadius,
	                                                                        pathChoice := #tempNextCmdIn.pathChoice,
	                                                                        circCenterPoint => #tempNextCmdIn.circleCenterPoint);
	          
	          IF (#tempRetValue <> 0) THEN
	            #LKinCtrl_OffsetContour.returnValue := #tempRetValue;
	            #LKinCtrl_OffsetContour."region" := #COFF_REGION_TYPE_RAD_COMP_NEXT_CMD_CIRC;
	            #LKinCtrl_OffsetContour.subBlockNumber := 35052;
	            #LKinCtrl_OffsetContour.internalNumber := 403;
	            RETURN;
	          END_IF;
	          
	        END_IF;
	        
	        //REGION todo
	        // 2019-03-07 - not necessary
	        (*
	        // ####
	        // Calculate circle paramters
	        #tempRetValue := "LKinCtrl_CalcCircTangOrthPathPlane"(circlePoint := #tempCurrentPoint,
	                                                              circleCenterPoint := #tempNextCmdIn.circleCenterPoint,
	                                                              pathPlane := #pathPlane,
	                                                              compDirection := #compensationDirection,
	                                                              pathChoice := #tempNextCmdIn.pathChoice,
	                                                              vUnitTangentialPathPlane => #tempNextCmdOut.tangentialUnitVecStart,
	                                                              vUnitOrthogonalPathPlane => #tempNextCmdOut.orthogonalUnitVecStart);
	        
	        IF (#tempRetValue <> 0) THEN
	          #LKinCtrl_OffsetContour.returnValue := #tempRetValue;
	          #LKinCtrl_OffsetContour."region" := #COFF_REGION_TYPE_RAD_COMP_LIN_CIRC;
	          #LKinCtrl_OffsetContour.subBlockNumber := 35056;
	          #LKinCtrl_OffsetContour.internalNumber := 404;
	          RETURN;
	        END_IF;
	        
	        // Scale othogonal vector with tool radius to get orthogonal shift
	        #tempNextCmdOut.orthogonalShiftStart := "LKinCtrl_VecScale"(vIn := #tempNextCmdOut.orthogonalUnitVecStart,
	                                                                    factor := #toolRadius);
	        
	        #tempNextCmdOut.startPointOrthShifted := "LKinCtrl_VecAdd"(vIn1 := #tempCurrentPoint,
	                                                                   vIn2 := #tempNextCmdOut.orthogonalShiftStart);
	        
	        *)
	        //END_REGION
	        
	        
	        // #############  N E X T   B U T   O N E   C M D   #############
	        // Check if next but one linear command has at least one component in path plane direction
	        #tempRetValue := "LKinCtrl_CalcVecDistancePathPlane"(vectorInA := #tempNextCmdIn.endPoint,
	                                                             vectorInB := #tempNextButOneCmdIn.endPoint,
	                                                             pathPlane := #pathPlane,
	                                                             distancePathPlane => #tempDistance1);
	        
	        IF (#tempRetValue <> 0) THEN
	          #LKinCtrl_OffsetContour.returnValue := #tempRetValue;
	          #LKinCtrl_OffsetContour."region" := #COFF_REGION_TYPE_RAD_COMP_CIRC_LIN;
	          #LKinCtrl_OffsetContour.subBlockNumber := 35055;
	          #LKinCtrl_OffsetContour.internalNumber := 405;
	          RETURN;
	        END_IF;
	        
	        // #############  N E X T   B U T   O N E   C M D   -  L I N E A R  #############
	        // Linear command must have at least a motion in direction of path plane, otherwise treat as command none!
	        IF (#tempNextButOneCmdOut.cmdType = "LKINCTRL_MC_MOVELINEARABS") AND (#tempDistance1 > 0.0) THEN
	          
	          REGION Next but one command LINEAR
	            // 2nd linear command point 2 to point 3
	            // Calculate tangential and orthogonal unit vector of direction (with respect to end point of circle)
	            #tempRetValue := "LKinCtrl_CalcLineTangOrthPathPlane"(pathPlane := #pathPlane,
	                                                                  compDirection := #compensationDirection,
	                                                                  vInFirst := #tempNextButOneCmdIn.endPoint,
	                                                                  vInSecond := #tempNextCmdIn.endPoint, // End point of circle
	                                                                  vUnitTangentialPathPlane => #tempNextButOneCmdOut.tangentialUnitVecStart,
	                                                                  vUnitOrthogonalPathPlane => #tempNextButOneCmdOut.orthogonalUnitVecStart);
	            
	            IF (#tempRetValue <> 0) THEN
	              #LKinCtrl_OffsetContour.returnValue := #tempRetValue;
	              #LKinCtrl_OffsetContour."region" := #COFF_REGION_TYPE_RAD_COMP_CIRC_LIN;
	              #LKinCtrl_OffsetContour.subBlockNumber := 35055;
	              #LKinCtrl_OffsetContour.internalNumber := 406;
	              RETURN;
	            END_IF;
	            
	            // Scale othogonal vector with tool radius to get orthogonal shift
	            #tempNextButOneCmdOut.orthogonalShiftStart := "LKinCtrl_VecScale"(vIn := #tempNextButOneCmdOut.orthogonalUnitVecStart,
	                                                                              factor := #toolRadius);
	            
	            // Scale tangential vector with tool radius to get tangential shift
	            #tempNextButOneCmdOut.tangentiaShiftStart := "LKinCtrl_VecScale"(vIn := #tempNextButOneCmdOut.tangentialUnitVecStart,
	                                                                             factor := #toolRadius);
	            
	            // Calculate orthogonal shifted next target coordinate
	            #tempNextButOneCmdOut.startPointOrthShifted := "LKinCtrl_VecAdd"(vIn1 := #tempNextCmdIn.endPoint, // Start coordinate next but one command
	                                                                             vIn2 := #tempNextButOneCmdOut.orthogonalShiftStart);
	            
	            // Calculate orthogonal and tangential shifted next target coordinate
	            #tempNextButOneCmdOut.startPointOrthTangShifted := "LKinCtrl_VecAdd"(vIn1 := #tempNextButOneCmdOut.startPointOrthShifted,
	                                                                                 vIn2 := #tempNextButOneCmdOut.tangentiaShiftStart);
	            
	            // ########## Intersection point of 1st circular and 2nd linear command  ##########
	            // Change center point to same level with start point
	            IF (#tempNextCmdIn.circleMode = "CM_BORDER") THEN
	              // ------------ Via an intermediate point and the end point ("CircMode" = 0) ------------
	              // 3D circle possible
	              
	              // Bring circle parameter to the same level as current point
	              #tempNextCmdEndPointLevelled := #tempNextCmdIn.endPoint;
	              #tempNextCmdIntermediatePointLevelled := #tempNextCmdIn.circleIntermediatePoint;
	              
	              
	              // Bring coordinates to same level as current point
	              #tempNextCmdStartPointOrhtShiftLevelled := #tempCurrentPointRadComp;// #tempNextCmdOut.startPointOrthShifted;
	              #tempNextButOneStartPointOrthShiftedLevelled := #tempNextButOneCmdOut.startPointOrthShifted;
	              #tempNextButOneCmdStartPointOrthTangShiftedLevelled := #tempNextButOneCmdOut.startPointOrthTangShifted;
	              
	              // Level parameters (third coordinate) with current point
	              CASE #pathPlane OF
	                "CP_XZ":
	                  #tempNextCmdEndPointLevelled.y := #tempCurrentPoint.y;
	                  #tempNextCmdIntermediatePointLevelled.y := #tempCurrentPoint.y;
	                  #tempNextCmdStartPointOrhtShiftLevelled.y := #tempCurrentPoint.y;
	                  #tempNextButOneStartPointOrthShiftedLevelled.y := #tempCurrentPoint.y;
	                  #tempNextButOneCmdStartPointOrthTangShiftedLevelled.y := #tempCurrentPoint.y;
	                  
	                "CP_YZ":
	                  #tempNextCmdEndPointLevelled.x := #tempCurrentPoint.x;
	                  #tempNextCmdIntermediatePointLevelled.x := #tempCurrentPoint.x;
	                  #tempNextCmdStartPointOrhtShiftLevelled.x := #tempCurrentPoint.x;
	                  #tempNextButOneStartPointOrthShiftedLevelled.x := #tempCurrentPoint.x;
	                  #tempNextButOneCmdStartPointOrthTangShiftedLevelled.x := #tempCurrentPoint.x;
	                  
	                "CP_XY":
	                  #tempNextCmdEndPointLevelled.z := #tempCurrentPoint.z;
	                  #tempNextCmdIntermediatePointLevelled.z := #tempCurrentPoint.z;
	                  #tempNextCmdStartPointOrhtShiftLevelled.z := #tempCurrentPoint.z;
	                  #tempNextButOneStartPointOrthShiftedLevelled.z := #tempCurrentPoint.z;
	                  #tempNextButOneCmdStartPointOrthTangShiftedLevelled.z := #tempCurrentPoint.z;
	                ELSE
	                  #LKinCtrl_OffsetContour.returnValue := #ERR_COFF_INTERNAL;
	                  #LKinCtrl_OffsetContour."region" := #COFF_REGION_TYPE_RAD_COMP_CIRC_LIN;
	                  #LKinCtrl_OffsetContour.internalNumber := 407;
	                  RETURN;
	              END_CASE;
	              
	              // Calculate new levelled circle center point
	              #tempRetValue := "LKinCtrl_CalcCircCenterByIntermediatePointAndEndPoint"(circleStartPoint := #tempCurrentPoint,
	                                                                                       circleEndPoint := #tempNextCmdEndPointLevelled,
	                                                                                       circleIntermediatePoint := #tempNextCmdIntermediatePointLevelled,
	                                                                                       pathPlane := #pathPlane,
	                                                                                       circleCenterPoint => #tempNextCmdOut.circleCenterPoint); // levelled
	              
	              IF (#tempRetValue <> 0) THEN
	                #LKinCtrl_OffsetContour.returnValue := #tempRetValue;
	                #LKinCtrl_OffsetContour."region" := #COFF_REGION_TYPE_RAD_COMP_NEXT_CMD_CIRC;
	                #LKinCtrl_OffsetContour.subBlockNumber := 35057;
	                #LKinCtrl_OffsetContour.internalNumber := 408;
	                RETURN;
	              END_IF;
	              
	              // Calculate modified radius - levelled
	              #tempNextCmdOut.circleRadius := "LKinCtrl_VecAbs"("LKinCtrl_VecSub"(vIn1 := #tempNextCmdStartPointOrhtShiftLevelled,
	                                                                                                                                    vIn2 := #tempNextCmdOut.circleCenterPoint));
	              
	              
	              
	              
	              #tempRetValue := "LKinCtrl_CalcLineCircleIntersectionPoint"(startPointLine := #tempNextButOneStartPointOrthShiftedLevelled,
	                                                                          endPointLine := #tempNextButOneCmdStartPointOrthTangShiftedLevelled,
	                                                                          circleCenter := #tempNextCmdOut.circleCenterPoint,
	                                                                          circleRadius := #tempNextCmdOut.circleRadius,
	                                                                          intersectionPointA => #tempPa,
	                                                                          intersectionPointB => #tempPb);
	              
	              // Relevel intersection point
	              CASE #pathPlane OF
	                "CP_XZ":
	                  #tempPa.y := #tempNextCmdIn.endPoint.y;
	                  #tempPb.y := #tempNextCmdIn.endPoint.y;
	                  
	                "CP_YZ":
	                  #tempPa.x := #tempNextCmdIn.endPoint.x;
	                  #tempPb.x := #tempNextCmdIn.endPoint.x;
	                  
	                "CP_XY":
	                  #tempPa.z := #tempNextCmdIn.endPoint.z;
	                  #tempPb.z := #tempNextCmdIn.endPoint.z;
	                ELSE
	                  #LKinCtrl_OffsetContour.returnValue := #ERR_COFF_INTERNAL;
	                  #LKinCtrl_OffsetContour."region" := #COFF_REGION_TYPE_RAD_COMP_CIRC_LIN;
	                  #LKinCtrl_OffsetContour.internalNumber := 409;
	                  RETURN;
	              END_CASE;
	              
	            ELSE
	              // 2D circle
	              // Calculate modified radius
	              #tempNextCmdOut.circleRadius := "LKinCtrl_VecAbs"("LKinCtrl_VecSub"(vIn1 := #tempCurrentPointRadComp,//#tempNextCmdOut.startPointOrthShifted,
	                                                                                                                                    vIn2 := #tempNextCmdIn.circleCenterPoint));
	              
	              #tempRetValue := "LKinCtrl_CalcLineCircleIntersectionPoint"(startPointLine := #tempNextButOneCmdOut.startPointOrthShifted,
	                                                                          endPointLine := #tempNextButOneCmdOut.startPointOrthTangShifted,
	                                                                          circleCenter := #tempNextCmdIn.circleCenterPoint,
	                                                                          circleRadius := #tempNextCmdOut.circleRadius,
	                                                                          intersectionPointA => #tempPa,
	                                                                          intersectionPointB => #tempPb);
	              
	              
	            END_IF;
	            
	            
	            IF (#tempRetValue <> 0) THEN
	              #LKinCtrl_OffsetContour.returnValue := #tempRetValue;
	              #LKinCtrl_OffsetContour."region" := #COFF_REGION_TYPE_RAD_COMP_CIRC_LIN;
	              #LKinCtrl_OffsetContour.subBlockNumber := 35061;
	              #LKinCtrl_OffsetContour.internalNumber := 410;
	              RETURN;
	            END_IF;
	            
	            // Two intersection points, use the one which is closer to the circle end point
	            #tempDistance1 := "LKinCtrl_VecAbs"("LKinCtrl_VecSub"(vIn1 := #tempNextCmdIn.endPoint, vIn2 := #tempPa));
	            #tempDistance2 := "LKinCtrl_VecAbs"("LKinCtrl_VecSub"(vIn1 := #tempNextCmdIn.endPoint, vIn2 := #tempPb));
	            
	            IF (#tempDistance1 < #tempDistance2) THEN
	              #tempNextCmdOut.endPoint := #tempPa;
	            ELSE
	              #tempNextCmdOut.endPoint := #tempPb;
	            END_IF;
	            
	          END_REGION
	          // #############  N E X T   B U T   O N E   C M D   -  C I R C U L A R #############
	        ELSIF (#tempNextButOneCmdOut.cmdType = "LKINCTRL_MC_MOVECIRCULARABS") THEN
	          REGION Next but one command CIRCULAR
	            // Distinguish between different circular modes
	            IF (#tempNextButOneCmdIn.circleMode = "CM_BORDER") THEN
	              // ------------ Via an intermediate point and the end point ("CircMode" = 0) ------------
	              
	              // Caluclate center point of circle with given start point, end point and intermediate point
	              #tempRetValue := "LKinCtrl_CalcCircCenterByIntermediatePointAndEndPoint"(circleStartPoint := #tempNextCmdIn.endPoint,
	                                                                                       circleEndPoint := #tempNextButOneCmdIn.endPoint,
	                                                                                       circleIntermediatePoint := #tempNextButOneCmdIn.circleIntermediatePoint,
	                                                                                       pathPlane := #pathPlane,
	                                                                                       circleCenterPoint => #tempNextButOneCmdIn.circleCenterPoint);
	              
	              IF (#tempRetValue <> 0) THEN
	                #LKinCtrl_OffsetContour.returnValue := #tempRetValue;
	                #LKinCtrl_OffsetContour."region" := #COFF_REGION_TYPE_RAD_COMP_CIRC_CIRC;
	                #LKinCtrl_OffsetContour.subBlockNumber := 35057;
	                #LKinCtrl_OffsetContour.internalNumber := 430;
	                RETURN;
	              END_IF;
	              
